C07319=1203.614,129.321,-51.756,-178.380,5.980,148.587
C07320=1203.610,129.570,-51.775,-178.377,5.982,148.587
C07321=1203.605,129.819,-51.796,-178.374,5.982,148.586
C07322=1203.600,130.069,-51.815,-178.372,5.984,148.586
C07323=1203.596,130.318,-51.836,-178.370,5.985,148.585
C07324=1203.591,130.567,-51.855,-178.366,5.986,148.585
C07325=1203.586,130.816,-51.875,-178.364,5.988,148.584
C07326=1203.581,131.065,-51.896,-178.361,5.989,148.584
C07327=1203.576,131.315,-51.916,-178.358,5.991,148.583
C07328=1203.572,131.563,-51.936,-178.356,5.992,148.583
C07329=1203.567,131.813,-51.956,-178.353,5.993,148.582
C07330=1203.563,132.062,-51.976,-178.351,5.994,148.582
C07331=1203.558,132.311,-51.997,-178.348,5.996,148.581
C07332=1203.552,132.560,-52.017,-178.346,5.996,148.581
C07333=1203.548,132.828,-52.039,-178.343,5.998,148.580
C07334=1203.542,133.098,-52.061,-178.340,5.999,148.580
C07335=1203.538,133.366,-52.082,-178.337,6.001,148.579
C07336=1203.532,133.635,-52.104,-178.334,6.003,148.579
C07337=1203.528,133.884,-52.124,-178.332,6.004,148.578
C07338=1203.523,134.133,-52.144,-178.329,6.005,148.578
C07339=1203.519,134.382,-52.164,-178.327,6.006,148.577
C07340=1203.513,134.631,-52.185,-178.324,6.008,148.577
C07341=1203.508,134.880,-52.205,-178.321,6.008,148.576
C07342=1203.504,135.129,-52.225,-178.319,6.010,148.576
C07343=1203.499,135.378,-52.245,-178.316,6.012,148.576
C07344=1203.494,135.628,-52.266,-178.313,6.013,148.575
C07345=1203.489,135.877,-52.286,-178.311,6.014,148.575
C07346=1203.485,136.126,-52.306,-178.309,6.015,148.574
C07347=1203.480,136.375,-52.327,-178.305,6.017,148.574
C07348=1203.475,136.624,-52.348,-178.303,6.018,148.573
C07349=1203.471,136.873,-52.368,-178.301,6.019,148.573
C07350=1203.466,137.123,-52.388,-178.297,6.021,148.572
C07351=1203.461,137.372,-52.409,-178.295,6.022,148.572
C07352=1203.456,137.621,-52.429,-178.293,6.024,148.571
C07353=1203.452,137.870,-52.450,-178.290,6.024,148.571
C07354=1203.447,138.119,-52.470,-178.287,6.026,148.570
C07355=1203.442,138.367,-52.490,-178.285,6.028,148.570
C07356=1203.437,138.616,-52.511,-178.282,6.028,148.569
C07357=1203.432,138.866,-52.531,-178.279,6.030,148.569
C07358=1203.427,139.115,-52.551,-178.277,6.031,148.569
C07359=1203.423,139.364,-52.572,-178.274,6.033,148.568
C07360=1203.418,139.613,-52.593,-178.271,6.034,148.568
C07361=1203.413,139.862,-52.613,-178.269,6.035,148.567
C07362=1203.408,140.112,-52.634,-178.266,6.037,148.567
C07363=1203.404,140.361,-52.655,-178.264,6.038,148.566
C07364=1203.399,140.610,-52.675,-178.261,6.040,148.566
C07365=1203.394,140.859,-52.696,-178.258,6.041,148.565
C07366=1203.390,141.108,-52.716,-178.256,6.042,148.565
C07367=1203.385,141.357,-52.737,-178.253,6.044,148.564
C07368=1203.381,141.607,-52.758,-178.251,6.046,148.564
C07369=1203.376,141.856,-52.778,-178.248,6.046,148.563
C07370=1203.371,142.105,-52.799,-178.245,6.048,148.563
C07371=1203.367,142.354,-52.820,-178.243,6.049,148.563
C07372=1203.362,142.603,-52.841,-178.240,6.050,148.562
C07373=1203.357,142.852,-52.861,-178.237,6.052,148.562
C07374=1203.352,143.101,-52.882,-178.235,6.053,148.561
C07375=1203.347,143.350,-52.902,-178.232,6.054,148.561
C07376=1203.342,143.599,-52.923,-178.229,6.056,148.560
C07377=1203.338,143.848,-52.944,-178.227,6.057,148.560
C07378=1203.333,144.098,-52.965,-178.225,6.059,148.559
C07379=1203.328,144.347,-52.985,-178.222,6.060,148.559
C07380=1203.323,144.595,-53.007,-178.219,6.061,148.558
C07381=1203.319,144.844,-53.027,-178.217,6.063,148.558
C07382=1203.314,145.093,-53.048,-178.214,6.064,148.557
C07383=1203.309,145.342,-53.068,-178.211,6.066,148.557
C07384=1203.305,145.592,-53.090,-178.209,6.067,148.557
C07385=1203.300,145.841,-53.110,-178.207,6.068,148.556
C07386=1203.295,146.091,-53.131,-178.204,6.070,148.556
C07387=1203.291,146.339,-53.152,-178.201,6.072,148.555
C07388=1203.286,146.588,-53.173,-178.199,6.073,148.555
C07389=1203.281,146.837,-53.193,-178.196,6.074,148.554
C07390=1203.276,147.086,-53.214,-178.193,6.076,148.554
C07391=1203.271,147.335,-53.236,-178.191,6.077,148.553
C07392=1203.268,147.585,-53.257,-178.188,6.079,148.553
C07393=1203.262,147.834,-53.278,-178.185,6.079,148.552
C07394=1203.258,148.083,-53.298,-178.183,6.081,148.552
C07395=1203.253,148.332,-53.320,-178.180,6.083,148.552
C07396=1203.248,148.581,-53.341,-178.178,6.084,148.551
C07397=1203.243,148.830,-53.361,-178.175,6.085,148.551
C07398=1203.238,149.079,-53.382,-178.172,6.087,148.550
C07399=1203.234,149.328,-53.404,-178.170,6.088,148.550
C07400=1203.230,149.577,-53.425,-178.167,6.090,148.550
C07401=1203.224,149.827,-53.446,-178.164,6.091,148.549
C07402=1203.219,150.075,-53.467,-178.162,6.092,148.549
C07403=1203.215,150.324,-53.488,-178.159,6.094,148.548
C07404=1203.210,150.573,-53.509,-178.157,6.096,148.548
C07405=1203.206,150.823,-53.531,-178.154,6.097,148.547
C07406=1203.201,151.072,-53.551,-178.151,6.098,148.547
C07407=1203.196,151.320,-53.573,-178.149,6.100,148.546
C07408=1203.191,151.570,-53.594,-178.146,6.102,148.546
C07409=1203.187,151.819,-53.614,-178.144,6.102,148.545
C07410=1203.182,152.068,-53.636,-178.141,6.104,148.545
C07411=1203.177,152.317,-53.657,-178.138,6.106,148.545
C07412=1203.172,152.566,-53.679,-178.136,6.107,148.544
C07413=1203.168,152.815,-53.699,-178.133,6.108,148.544
C07414=1203.163,153.063,-53.721,-178.130,6.110,148.543
C07415=1203.159,153.313,-53.742,-178.128,6.111,148.543
C07416=1203.154,153.562,-53.764,-178.125,6.113,148.543
C07417=1203.149,153.811,-53.784,-178.122,6.114,148.542
C07418=1203.144,154.060,-53.805,-178.120,6.115,148.542
C07419=1203.140,154.310,-53.827,-178.118,6.117,148.541
C07420=1203.135,154.558,-53.849,-178.115,6.119,148.541
C07421=1203.130,154.807,-53.869,-178.112,6.120,148.540
C07422=1203.126,155.056,-53.891,-178.110,6.121,148.540
C07423=1203.121,155.306,-53.912,-178.107,6.123,148.539
C07424=1203.116,155.554,-53.934,-178.104,6.125,148.539
C07425=1203.111,155.804,-53.955,-178.102,6.126,148.539
C07426=1203.107,156.053,-53.977,-178.099,6.127,148.538
C07427=1203.102,156.302,-53.997,-178.096,6.129,148.538
C07428=1203.097,156.551,-54.019,-178.094,6.131,148.537
C07429=1203.093,156.799,-54.041,-178.092,6.132,148.537
C07430=1203.088,157.049,-54.062,-178.089,6.134,148.537
C07431=1203.083,157.298,-54.084,-178.086,6.135,148.536
C07432=1203.078,157.546,-54.105,-178.084,6.136,148.536
C07433=1203.074,157.796,-54.127,-178.081,6.138,148.535
C07434=1203.070,158.045,-54.148,-178.078,6.140,148.535
C07435=1203.065,158.293,-54.170,-178.075,6.141,148.534
C07436=1203.060,158.543,-54.191,-178.073,6.142,148.534
C07437=1203.055,158.812,-54.215,-178.070,6.144,148.533
C07438=1203.050,159.080,-54.237,-178.068,6.146,148.533
C07439=1203.044,159.350,-54.261,-178.064,6.147,148.533
C07440=1203.040,159.618,-54.284,-178.062,6.149,148.532
C07441=1203.035,159.868,-54.305,-178.059,6.151,148.532
C07442=1203.030,160.117,-54.327,-178.056,6.152,148.531
C07443=1203.025,160.365,-54.349,-178.054,6.153,148.531
C07444=1203.021,160.615,-54.371,-178.051,6.155,148.530
C07445=1203.016,160.864,-54.392,-178.049,6.157,148.530
C07446=1203.012,161.113,-54.414,-178.046,6.158,148.530
C07447=1203.007,161.362,-54.436,-178.043,6.159,148.529
C07448=1203.002,161.611,-54.457,-178.041,6.161,148.529
C07449=1202.998,161.860,-54.479,-178.038,6.163,148.528
C07450=1202.992,162.109,-54.500,-178.035,6.164,148.528
C07451=1202.988,162.359,-54.522,-178.033,6.165,148.528
C07452=1202.983,162.607,-54.544,-178.030,6.167,148.527
C07453=1202.978,162.856,-54.566,-178.027,6.169,148.527
C07454=1202.974,163.105,-54.588,-178.025,6.170,148.526
C07455=1202.969,163.354,-54.609,-178.023,6.171,148.526
C07456=1202.965,163.603,-54.631,-178.020,6.173,148.525
C07457=1202.960,163.852,-54.653,-178.017,6.175,148.525
C07458=1202.955,164.100,-54.675,-178.015,6.177,148.525
C07459=1202.951,164.350,-54.696,-178.012,6.177,148.524
C07460=1202.946,164.599,-54.718,-178.009,6.179,148.524
C07461=1202.942,164.848,-54.740,-178.007,6.181,148.523
C07462=1202.936,165.097,-54.762,-178.004,6.183,148.523
C07463=1202.932,165.347,-54.784,-178.002,6.184,148.523
C07464=1202.927,165.595,-54.806,-177.999,6.186,148.522
C07465=1202.923,165.845,-54.828,-177.996,6.187,148.522
C07466=1202.918,166.093,-54.850,-177.993,6.189,148.521
C07467=1202.913,166.342,-54.871,-177.991,6.191,148.521
C07468=1202.909,166.591,-54.893,-177.989,6.192,148.521
C07469=1202.904,166.840,-54.915,-177.986,6.193,148.520
C07470=1202.899,167.089,-54.937,-177.983,6.195,148.520
C07471=1202.894,167.338,-54.959,-177.981,6.197,148.519
C07472=1202.890,167.587,-54.982,-177.978,6.198,148.519
C07473=1202.885,167.836,-55.004,-177.975,6.199,148.518
C07474=1202.881,168.085,-55.026,-177.973,6.201,148.518
C07475=1202.876,168.334,-55.048,-177.970,6.203,148.518
C07476=1202.872,168.583,-55.070,-177.967,6.205,148.517
C07477=1202.866,168.832,-55.092,-177.965,6.206,148.517
C07478=1202.862,169.081,-55.114,-177.963,6.208,148.517
C07479=1202.857,169.330,-55.136,-177.959,6.209,148.516
C07480=1202.853,169.579,-55.158,-177.957,6.211,148.516
C07481=1202.848,169.827,-55.180,-177.954,6.213,148.515
C07482=1202.843,170.077,-55.203,-177.952,6.214,148.515
C07483=1202.838,170.326,-55.224,-177.949,6.215,148.515
C07484=1202.834,170.575,-55.246,-177.947,6.217,148.514
C07485=1202.830,170.824,-55.268,-177.944,6.219,148.514
C07486=1202.824,171.073,-55.291,-177.941,6.221,148.513
C07487=1202.820,171.322,-55.314,-177.939,6.222,148.513
C07488=1202.815,171.571,-55.335,-177.936,6.223,148.513
C07489=1202.810,171.820,-55.358,-177.933,6.225,148.512
C07490=1202.806,172.068,-55.380,-177.931,6.227,148.512
C07491=1202.801,172.318,-55.402,-177.928,6.229,148.511
C07492=1202.796,172.566,-55.424,-177.925,6.231,148.511
C07493=1202.791,172.816,-55.447,-177.923,6.232,148.511
C07494=1202.787,173.065,-55.469,-177.921,6.233,148.510
C07495=1202.783,173.313,-55.491,-177.918,6.235,148.510
C07496=1202.778,173.563,-55.514,-177.915,6.237,148.509
C07497=1202.773,173.811,-55.536,-177.912,6.238,148.509
C07498=1202.769,174.060,-55.558,-177.909,6.240,148.509
C07499=1202.764,174.310,-55.581,-177.907,6.241,148.508
C07500=1202.759,174.558,-55.603,-177.905,6.243,148.508
C07501=1202.755,174.807,-55.625,-177.902,6.245,148.508
C07502=1202.749,175.056,-55.648,-177.899,6.247,148.507
C07503=1202.745,175.305,-55.670,-177.897,6.248,148.507
C07504=1202.740,175.555,-55.693,-177.894,6.250,148.506
C07505=1202.736,175.803,-55.715,-177.892,6.251,148.506
C07506=1202.732,176.052,-55.737,-177.889,6.253,148.506
C07507=1202.727,176.301,-55.761,-177.886,6.254,148.505
C07508=1202.722,176.550,-55.782,-177.883,6.256,148.505
C07509=1202.717,176.799,-55.805,-177.881,6.258,148.504
C07510=1202.713,177.048,-55.828,-177.878,6.260,148.504
C07511=1202.708,177.297,-55.850,-177.876,6.261,148.504
C07512=1202.703,177.546,-55.873,-177.873,6.263,148.503
C07513=1202.699,177.795,-55.895,-177.871,6.264,148.503
C07514=1202.694,178.043,-55.918,-177.868,6.266,148.503
C07515=1202.690,178.293,-55.940,-177.865,6.268,148.502
C07516=1202.685,178.542,-55.963,-177.863,6.270,148.502
C07517=1202.680,178.790,-55.986,-177.860,6.272,148.502
C07518=1202.675,179.039,-56.008,-177.858,6.273,148.501
C07519=1202.671,179.288,-56.031,-177.855,6.274,148.501
C07520=1202.666,179.537,-56.053,-177.852,6.276,148.500
C07521=1202.662,179.786,-56.076,-177.849,6.278,148.500
C07522=1202.657,180.035,-56.099,-177.847,6.280,148.499
C07523=1202.653,180.284,-56.122,-177.844,6.281,148.499
C07524=1202.647,180.532,-56.145,-177.841,6.283,148.499
C07525=1202.643,180.782,-56.167,-177.839,6.285,148.498
C07526=1202.639,181.031,-56.190,-177.837,6.286,148.498
C07527=1202.635,181.280,-56.213,-177.834,6.288,148.498
C07528=1202.629,181.528,-56.235,-177.831,6.290,148.497
C07529=1202.625,181.777,-56.258,-177.829,6.291,148.497
C07530=1202.620,182.026,-56.281,-177.826,6.293,148.497
C07531=1202.615,182.276,-56.304,-177.823,6.295,148.496
C07532=1202.611,182.524,-56.326,-177.821,6.297,148.496
C07533=1202.606,182.773,-56.350,-177.818,6.299,148.496
C07534=1202.602,183.022,-56.372,-177.815,6.300,148.495
C07535=1202.597,183.271,-56.395,-177.813,6.301,148.495
C07536=1202.592,183.519,-56.417,-177.811,6.303,148.494
C07537=1202.588,183.768,-56.441,-177.808,6.305,148.494
C07538=1202.583,184.017,-56.464,-177.805,6.307,148.494
C07539=1202.579,184.267,-56.486,-177.803,6.309,148.493
C07540=1202.574,184.516,-56.509,-177.800,6.310,148.493
C07541=1202.569,184.786,-56.535,-177.797,6.312,148.492
C07542=1202.564,185.055,-56.559,-177.794,6.314,148.492
C07543=1202.559,185.325,-56.584,-177.792,6.316,148.492
C07544=1202.554,185.594,-56.608,-177.789,6.317,148.491
C07545=1202.549,185.843,-56.631,-177.786,6.319,148.491
C07546=1202.544,186.092,-56.655,-177.784,6.321,148.491
C07547=1202.540,186.341,-56.678,-177.781,6.323,148.490
C07548=1202.536,186.589,-56.701,-177.778,6.325,148.490
C07549=1202.531,186.838,-56.724,-177.776,6.326,148.490
C07550=1202.526,187.087,-56.748,-177.773,6.328,148.489
C07551=1202.522,187.335,-56.770,-177.770,6.330,148.489
C07552=1202.517,187.584,-56.793,-177.768,6.332,148.489
C07553=1202.512,187.834,-56.816,-177.765,6.334,148.488
C07554=1202.507,188.083,-56.839,-177.762,6.335,148.488
C07555=1202.503,188.332,-56.862,-177.760,6.337,148.488
C07556=1202.499,188.581,-56.886,-177.758,6.338,148.487
C07557=1202.494,188.830,-56.909,-177.755,6.340,148.487
C07558=1202.489,189.078,-56.932,-177.752,6.342,148.486
C07559=1202.485,189.327,-56.955,-177.750,6.344,148.486
C07560=1202.480,189.576,-56.978,-177.747,6.346,148.486
C07561=1202.475,189.825,-57.001,-177.744,6.347,148.485
C07562=1202.471,190.074,-57.025,-177.742,6.349,148.485
C07563=1202.466,190.323,-57.048,-177.739,6.351,148.485
C07564=1202.461,190.572,-57.071,-177.736,6.353,148.484
C07565=1202.458,190.820,-57.095,-177.734,6.355,148.484
C07566=1202.453,191.069,-57.118,-177.731,6.356,148.484
C07567=1202.448,191.318,-57.141,-177.728,6.358,148.483
C07568=1202.443,191.567,-57.165,-177.726,6.360,148.483
C07569=1202.438,191.816,-57.188,-177.723,6.362,148.483
C07570=1202.433,192.065,-57.211,-177.720,6.364,148.482
C07571=1202.429,192.313,-57.234,-177.718,6.365,148.482
C07572=1202.425,192.562,-57.257,-177.715,6.367,148.482
C07573=1202.420,192.811,-57.281,-177.712,6.369,148.481
C07574=1202.416,193.060,-57.305,-177.710,6.370,148.481
C07575=1202.411,193.309,-57.328,-177.708,6.372,148.480
C07576=1202.406,193.558,-57.352,-177.705,6.374,148.480
C07577=1202.402,193.807,-57.375,-177.702,6.376,148.480
C07578=1202.397,194.056,-57.398,-177.700,6.377,148.479
C07579=1202.392,194.304,-57.422,-177.697,6.379,148.479
C07580=1202.388,194.553,-57.446,-177.694,6.381,148.479
C07581=1202.383,194.802,-57.469,-177.692,6.383,148.478
C07582=1202.378,195.052,-57.492,-177.689,6.385,148.478
C07583=1202.374,195.300,-57.517,-177.686,6.386,148.478
C07584=1202.369,195.549,-57.540,-177.684,6.388,148.477
C07585=1202.365,195.798,-57.563,-177.681,6.390,148.477
C07586=1202.361,196.047,-57.586,-177.678,6.392,148.477
C07587=1202.356,196.295,-57.610,-177.676,6.394,148.476
C07588=1202.352,196.544,-57.633,-177.673,6.396,148.476
C07589=1202.347,196.793,-57.657,-177.671,6.397,148.476
C07590=1202.342,197.042,-57.681,-177.668,6.399,148.475
C07591=1202.338,197.291,-57.704,-177.665,6.401,148.475
C07592=1202.332,197.540,-57.728,-177.663,6.403,148.475
C07593=1202.328,197.788,-57.752,-177.660,6.405,148.474
C07594=1202.323,198.037,-57.776,-177.658,6.407,148.474
C07595=1202.319,198.286,-57.800,-177.655,6.409,148.474
C07596=1202.314,198.535,-57.823,-177.652,6.410,148.473
C07597=1202.309,198.784,-57.846,-177.650,6.412,148.473
C07598=1202.305,199.032,-57.870,-177.647,6.414,148.473
C07599=1202.300,199.281,-57.894,-177.644,6.416,148.472
C07600=1202.296,199.530,-57.918,-177.642,6.418,148.472
C07601=1202.291,199.779,-57.941,-177.639,6.420,148.472
C07602=1202.287,200.027,-57.965,-177.637,6.421,148.471
C07603=1202.283,200.277,-57.989,-177.634,6.423,148.471
C07604=1202.278,200.525,-58.013,-177.631,6.425,148.471
C07605=1202.273,200.775,-58.037,-177.629,6.427,148.470
C07606=1202.268,201.023,-58.061,-177.626,6.429,148.470
C07607=1202.264,201.272,-58.085,-177.624,6.431,148.470
C07608=1202.259,201.521,-58.109,-177.621,6.433,148.469
C07609=1202.255,201.770,-58.132,-177.618,6.434,148.469
C07610=1202.250,202.018,-58.156,-177.616,6.436,148.469
C07611=1202.246,202.267,-58.179,-177.613,6.438,148.468
C07612=1202.240,202.516,-58.204,-177.610,6.440,148.468
C07613=1202.237,202.765,-58.229,-177.608,6.442,148.468
C07614=1202.232,203.014,-58.252,-177.605,6.444,148.467
C07615=1202.228,203.262,-58.276,-177.603,6.445,148.467
C07616=1202.223,203.511,-58.300,-177.600,6.447,148.467
C07617=1202.218,203.760,-58.324,-177.597,6.449,148.466
C07618=1202.213,204.008,-58.348,-177.595,6.451,148.466
C07619=1202.209,204.258,-58.372,-177.592,6.453,148.466
C07620=1202.205,204.507,-58.396,-177.590,6.455,148.466
C07621=1202.200,204.755,-58.420,-177.587,6.457,148.465
C07622=1202.195,205.004,-58.445,-177.584,6.458,148.465
C07623=1202.191,205.253,-58.468,-177.582,6.460,148.465
C07624=1202.186,205.501,-58.492,-177.579,6.462,148.464
C07625=1202.182,205.750,-58.516,-177.576,6.465,148.464
C07626=1202.177,206.000,-58.540,-177.573,6.467,148.464
C07627=1202.173,206.248,-58.565,-177.571,6.469,148.463
C07628=1202.168,206.496,-58.589,-177.568,6.471,148.463
C07629=1202.163,206.745,-58.613,-177.566,6.472,148.463
C07630=1202.159,206.995,-58.637,-177.563,6.474,148.462
C07631=1202.155,207.243,-58.661,-177.561,6.476,148.462
C07632=1202.149,207.492,-58.686,-177.558,6.478,148.462
C07633=1202.145,207.741,-58.710,-177.555,6.480,148.461
C07634=1202.141,207.989,-58.734,-177.553,6.481,148.461
C07635=1202.136,208.238,-58.759,-177.550,6.484,148.461
C07636=1202.131,208.487,-58.782,-177.548,6.485,148.461
C07637=1202.127,208.736,-58.806,-177.545,6.487,148.460
C07638=1202.122,208.985,-58.831,-177.542,6.489,148.460
C07639=1202.118,209.234,-58.855,-177.540,6.491,148.460
C07640=1202.114,209.482,-58.880,-177.537,6.493,148.459
C07641=1202.109,209.731,-58.904,-177.535,6.495,148.459
C07642=1202.104,209.979,-58.928,-177.532,6.498,148.459
C07643=1202.100,210.229,-58.953,-177.529,6.499,148.459
C07644=1202.095,210.477,-58.977,-177.527,6.501,148.458
C07645=1202.090,210.748,-59.003,-177.524,6.503,148.458
C07646=1202.085,211.018,-59.030,-177.521,6.505,148.458
C07647=1202.080,211.289,-59.057,-177.518,6.508,148.457
C07648=1202.076,211.559,-59.083,-177.515,6.509,148.457
C07649=1202.071,211.807,-59.108,-177.513,6.511,148.457
C07650=1202.066,212.056,-59.132,-177.510,6.513,148.456
C07651=1202.062,212.305,-59.157,-177.507,6.515,148.456
C07652=1202.057,212.554,-59.181,-177.505,6.517,148.456
C07653=1202.052,212.802,-59.206,-177.502,6.520,148.455
C07654=1202.048,213.052,-59.230,-177.499,6.521,148.455
C07655=1202.043,213.300,-59.255,-177.497,6.523,148.455
C07656=1202.039,213.549,-59.279,-177.494,6.525,148.454
C07657=1202.034,213.798,-59.304,-177.491,6.527,148.454
C07658=1202.030,214.046,-59.328,-177.489,6.529,148.454
C07659=1202.025,214.295,-59.353,-177.487,6.531,148.454
C07660=1202.021,214.544,-59.378,-177.484,6.533,148.453
C07661=1202.016,214.792,-59.403,-177.481,6.535,148.453
C07662=1202.012,215.041,-59.427,-177.479,6.536,148.453
C07663=1202.007,215.290,-59.452,-177.476,6.539,148.452
C07664=1202.002,215.539,-59.476,-177.473,6.541,148.452
C07665=1201.998,215.788,-59.501,-177.471,6.543,148.452
C07666=1201.993,216.036,-59.526,-177.468,6.545,148.452
C07667=1201.989,216.285,-59.550,-177.465,6.547,148.451
C07668=1201.985,216.534,-59.575,-177.463,6.549,148.451
C07669=1201.980,216.782,-59.599,-177.460,6.550,148.451
C07670=1201.975,217.031,-59.624,-177.458,6.553,148.450
C07671=1201.971,217.280,-59.650,-177.455,6.554,148.450
C07672=1201.966,217.528,-59.674,-177.452,6.557,148.450
C07673=1201.962,217.778,-59.699,-177.449,6.559,148.449
C07674=1201.957,218.026,-59.724,-177.447,6.561,148.449
C07675=1201.953,218.274,-59.748,-177.445,6.563,148.449
C07676=1201.948,218.524,-59.773,-177.442,6.565,148.449
C07677=1201.943,218.772,-59.798,-177.439,6.567,148.448
C07678=1201.939,219.021,-59.823,-177.437,6.568,148.448
C07679=1201.934,219.270,-59.848,-177.434,6.570,148.448
C07680=1201.930,219.519,-59.873,-177.431,6.573,148.448
C07681=1201.926,219.767,-59.898,-177.429,6.575,148.447
C07682=1201.921,220.016,-59.923,-177.426,6.577,148.447
C07683=1201.916,220.264,-59.948,-177.423,6.579,148.447
C07684=1201.913,220.514,-59.973,-177.421,6.581,148.446
C07685=1201.907,220.762,-59.997,-177.419,6.583,148.446
C07686=1201.903,221.010,-60.023,-177.416,6.584,148.446
C07687=1201.898,221.260,-60.048,-177.413,6.586,148.446
C07688=1201.894,221.508,-60.072,-177.410,6.589,148.445
C07689=1201.889,221.757,-60.097,-177.408,6.591,148.445
C07690=1201.885,222.005,-60.123,-177.405,6.593,148.445
C07691=1201.880,222.255,-60.148,-177.403,6.595,148.444
C07692=1201.876,222.502,-60.173,-177.400,6.597,148.444
C07693=1201.872,222.752,-60.198,-177.398,6.599,148.444
C07694=1201.867,223.000,-60.223,-177.395,6.601,148.444
C07695=1201.862,223.249,-60.248,-177.392,6.603,148.443
C07696=1201.857,223.497,-60.274,-177.389,6.605,148.443
C07697=1201.854,223.747,-60.298,-177.387,6.607,148.443
C07698=1201.849,223.995,-60.323,-177.385,6.609,148.443
C07699=1201.844,224.244,-60.348,-177.382,6.611,148.442
C07700=1201.840,224.493,-60.374,-177.379,6.613,148.442
C07701=1201.835,224.741,-60.400,-177.377,6.616,148.442
C07702=1201.831,224.990,-60.425,-177.374,6.618,148.442
C07703=1201.827,225.238,-60.449,-177.371,6.619,148.441
C07704=1201.822,225.488,-60.474,-177.369,6.621,148.441
C07705=1201.817,225.736,-60.500,-177.367,6.623,148.441
C07706=1201.813,225.984,-60.526,-177.364,6.625,148.441
C07707=1201.808,226.233,-60.550,-177.361,6.627,148.440
C07708=1201.804,226.482,-60.576,-177.358,6.630,148.440
C07709=1201.799,226.731,-60.602,-177.356,6.632,148.440
C07710=1201.794,226.980,-60.626,-177.353,6.634,148.439
C07711=1201.790,227.228,-60.652,-177.351,6.636,148.439
C07712=1201.786,227.476,-60.677,-177.348,6.638,148.439
C07713=1201.782,227.725,-60.703,-177.346,6.640,148.439
C07714=1201.777,227.974,-60.728,-177.343,6.642,148.438
C07715=1201.772,228.222,-60.753,-177.340,6.644,148.438
C07716=1201.768,228.471,-60.779,-177.338,6.646,148.438
C07717=1201.763,228.719,-60.804,-177.335,6.648,148.438
C07718=1201.759,228.969,-60.829,-177.333,6.650,148.437
C07719=1201.755,229.218,-60.855,-177.330,6.653,148.437
C07720=1201.750,229.466,-60.880,-177.327,6.655,148.437
C07721=1201.745,229.715,-60.906,-177.325,6.657,148.437
C07722=1201.741,229.963,-60.932,-177.322,6.659,148.437
C07723=1201.736,230.212,-60.957,-177.320,6.661,148.436
C07724=1201.732,230.461,-60.982,-177.317,6.662,148.436
C07725=1201.727,230.709,-61.008,-177.314,6.665,148.436
C07726=1201.723,230.958,-61.033,-177.312,6.667,148.435
C07727=1201.719,231.207,-61.059,-177.309,6.669,148.435
C07728=1201.714,231.455,-61.085,-177.307,6.671,148.435
C07729=1201.710,231.703,-61.110,-177.304,6.673,148.435
C07730=1201.705,231.952,-61.136,-177.301,6.676,148.434
C07731=1201.700,232.201,-61.162,-177.299,6.678,148.434
C07732=1201.696,232.450,-61.188,-177.296,6.680,148.434
C07733=1201.691,232.699,-61.213,-177.294,6.682,148.434
C07734=1201.687,232.948,-61.239,-177.291,6.683,148.433
C07735=1201.682,233.196,-61.264,-177.288,6.686,148.433
C07736=1201.678,233.445,-61.290,-177.286,6.688,148.433
C07737=1201.674,233.693,-61.316,-177.283,6.690,148.433
C07738=1201.669,233.942,-61.341,-177.281,6.692,148.433
C07739=1201.664,234.190,-61.367,-177.278,6.694,148.432
C07740=1201.660,234.439,-61.394,-177.275,6.697,148.432
C07741=1201.655,234.687,-61.419,-177.273,6.699,148.432
C07742=1201.651,234.936,-61.445,-177.270,6.701,148.432
C07743=1201.647,235.185,-61.471,-177.268,6.703,148.431
C07744=1201.642,235.433,-61.496,-177.266,6.705,148.431
C07745=1201.637,235.681,-61.522,-177.262,6.708,148.431
C07746=1201.633,235.931,-61.548,-177.260,6.710,148.431
C07747=1201.628,236.179,-61.574,-177.258,6.712,148.430
C07748=1201.624,236.428,-61.600,-177.255,6.713,148.430
C07749=1201.619,236.699,-61.628,-177.252,6.716,148.430
C07750=1201.614,236.971,-61.656,-177.250,6.718,148.430
C07751=1201.610,237.243,-61.684,-177.246,6.721,148.429
C07752=1201.604,237.513,-61.713,-177.244,6.723,148.429
C07753=1201.600,237.762,-61.739,-177.241,6.726,148.429
C07754=1201.596,238.011,-61.765,-177.238,6.728,148.429
C07755=1201.591,238.260,-61.790,-177.236,6.729,148.428
C07756=1201.587,238.508,-61.817,-177.234,6.732,148.428
C07757=1201.582,238.756,-61.843,-177.230,6.734,148.428
C07758=1201.578,239.005,-61.868,-177.228,6.736,148.428
C07759=1201.573,239.254,-61.894,-177.226,6.738,148.428
C07760=1201.569,239.503,-61.921,-177.223,6.740,148.427
C07761=1201.564,239.751,-61.947,-177.221,6.742,148.427
C07762=1201.560,239.999,-61.972,-177.218,6.745,148.427
C07763=1201.555,240.248,-61.999,-177.215,6.747,148.427
C07764=1201.551,240.497,-62.025,-177.213,6.749,148.426
C07765=1201.547,240.746,-62.051,-177.210,6.751,148.426
C07766=1201.542,240.994,-62.078,-177.207,6.754,148.426
C07767=1201.538,241.243,-62.104,-177.205,6.756,148.426
C07768=1201.533,241.491,-62.129,-177.203,6.758,148.426
C07769=1201.528,241.739,-62.156,-177.200,6.760,148.425
C07770=1201.524,241.988,-62.182,-177.197,6.762,148.425
C07771=1201.519,242.237,-62.208,-177.195,6.764,148.425
C07772=1201.515,242.486,-62.235,-177.192,6.766,148.425
C07773=1201.511,242.734,-62.261,-177.189,6.769,148.425
C07774=1201.506,242.983,-62.288,-177.187,6.771,148.424
C07775=1201.502,243.232,-62.313,-177.184,6.773,148.424
C07776=1201.497,243.480,-62.340,-177.182,6.775,148.424
C07777=1201.492,243.728,-62.366,-177.179,6.778,148.424
C07778=1201.489,243.976,-62.392,-177.177,6.780,148.423
C07779=1201.484,244.226,-62.419,-177.174,6.782,148.423
C07780=1201.480,244.474,-62.445,-177.172,6.784,148.423
C07781=1201.475,244.723,-62.471,-177.169,6.787,148.423
C07782=1201.471,244.971,-62.498,-177.166,6.789,148.422
C07783=1201.466,245.220,-62.524,-177.164,6.791,148.422
C07784=1201.462,245.468,-62.551,-177.161,6.793,148.422
C07785=1201.457,245.718,-62.577,-177.159,6.796,148.422
C07786=1201.453,245.966,-62.604,-177.156,6.797,148.422
C07787=1201.448,246.214,-62.631,-177.154,6.800,148.422
C07788=1201.444,246.463,-62.656,-177.151,6.802,148.421
C07789=1201.440,246.711,-62.683,-177.148,6.804,148.421
C07790=1201.435,246.960,-62.709,-177.146,6.806,148.421
C07791=1201.430,247.208,-62.736,-177.143,6.809,148.421
C07792=1201.426,247.456,-62.762,-177.140,6.811,148.421
C07793=1201.421,247.705,-62.789,-177.138,6.813,148.420
C07794=1201.417,247.954,-62.815,-177.136,6.815,148.420
C07795=1201.413,248.202,-62.842,-177.132,6.818,148.420
C07796=1201.408,248.451,-62.869,-177.130,6.820,148.420
C07797=1201.404,248.699,-62.895,-177.128,6.822,148.419
C07798=1201.399,248.948,-62.922,-177.125,6.825,148.419
C07799=1201.395,249.197,-62.948,-177.122,6.827,148.419
C07800=1201.390,249.445,-62.975,-177.120,6.829,148.419
C07801=1201.385,249.694,-63.002,-177.117,6.832,148.419
C07802=1201.382,249.942,-63.028,-177.115,6.834,148.419
C07803=1201.377,250.190,-63.055,-177.112,6.836,148.418
C07804=1201.373,250.439,-63.081,-177.110,6.838,148.418
C07805=1201.368,250.688,-63.108,-177.107,6.840,148.418
C07806=1201.363,250.936,-63.135,-177.105,6.843,148.418
C07807=1201.360,251.185,-63.162,-177.102,6.844,148.418
C07808=1201.355,251.434,-63.189,-177.099,6.847,148.418
C07809=1201.350,251.683,-63.216,-177.097,6.849,148.417
C07810=1201.347,251.931,-63.242,-177.095,6.851,148.417
C07811=1201.342,252.179,-63.269,-177.091,6.854,148.417
C07812=1201.337,252.428,-63.296,-177.089,6.856,148.417
C07813=1201.333,252.676,-63.323,-177.087,6.858,148.416
C07814=1201.329,252.924,-63.350,-177.084,6.861,148.416
C07815=1201.324,253.173,-63.377,-177.081,6.863,148.416
C07816=1201.319,253.421,-63.404,-177.079,6.865,148.416
C07817=1201.315,253.670,-63.430,-177.076,6.868,148.416
C07818=1201.311,253.918,-63.457,-177.074,6.870,148.416
C07819=1201.306,254.167,-63.484,-177.071,6.872,148.415
C07820=1201.301,254.415,-63.511,-177.068,6.875,148.415
C07821=1201.298,254.664,-63.538,-177.066,6.877,148.415
C07822=1201.293,254.913,-63.565,-177.064,6.879,148.415
C07823=1201.289,255.161,-63.592,-177.061,6.882,148.415
C07824=1201.284,255.410,-63.619,-177.058,6.884,148.415
C07825=1201.279,255.658,-63.647,-177.056,6.886,148.414
C07826=1201.276,255.906,-63.673,-177.053,6.889,148.414
C07827=1201.271,256.155,-63.700,-177.051,6.891,148.414
C07828=1201.266,256.403,-63.727,-177.048,6.894,148.414
C07829=1201.262,256.652,-63.755,-177.046,6.896,148.414
C07830=1201.258,256.901,-63.782,-177.043,6.898,148.413
C07831=1201.253,257.149,-63.809,-177.040,6.901,148.413
C07832=1201.249,257.398,-63.835,-177.038,6.902,148.413
C07833=1201.244,257.646,-63.862,-177.035,6.905,148.413
C07834=1201.240,257.895,-63.889,-177.032,6.907,148.413
C07835=1201.236,258.143,-63.917,-177.030,6.909,148.413
C07836=1201.231,258.392,-63.944,-177.028,6.912,148.413
C07837=1201.227,258.640,-63.972,-177.025,6.914,148.412
C07838=1201.222,258.889,-63.999,-177.023,6.916,148.412
C07839=1201.217,259.137,-64.026,-177.019,6.919,148.412
C07840=1201.214,259.385,-64.053,-177.017,6.921,148.412
C07841=1201.210,259.634,-64.080,-177.015,6.923,148.412
C07842=1201.205,259.882,-64.107,-177.012,6.926,148.411
C07843=1201.200,260.131,-64.134,-177.010,6.928,148.411
C07844=1201.196,260.379,-64.162,-177.007,6.930,148.411
C07845=1201.192,260.628,-64.190,-177.004,6.933,148.411
C07846=1201.187,260.876,-64.217,-177.002,6.935,148.411
C07847=1201.183,261.125,-64.244,-176.999,6.938,148.411
C07848=1201.178,261.373,-64.271,-176.997,6.940,148.411
C07849=1201.174,261.621,-64.299,-176.994,6.942,148.410
C07850=1201.170,261.871,-64.326,-176.992,6.945,148.410
C07851=1201.165,262.118,-64.354,-176.989,6.947,148.410
C07852=1201.161,262.367,-64.381,-176.986,6.950,148.410
C07853=1201.156,262.640,-64.412,-176.984,6.952,148.410
C07854=1201.151,262.913,-64.441,-176.981,6.955,148.410
C07855=1201.146,263.185,-64.472,-176.978,6.958,148.409
C07856=1201.141,263.458,-64.502,-176.975,6.961,148.409
C07857=1201.137,263.707,-64.529,-176.973,6.962,148.409
C07858=1201.132,263.955,-64.557,-176.970,6.965,148.409
C07859=1201.128,264.203,-64.584,-176.968,6.968,148.409
C07860=1201.124,264.453,-64.612,-176.965,6.969,148.409
C07861=1201.119,264.700,-64.639,-176.962,6.972,148.408
C07862=1201.115,264.949,-64.666,-176.960,6.975,148.408
C07863=1201.111,265.197,-64.695,-176.958,6.976,148.408
C07864=1201.106,265.446,-64.722,-176.955,6.979,148.408
C07865=1201.102,265.694,-64.749,-176.952,6.981,148.408
C07866=1201.097,265.942,-64.776,-176.950,6.984,148.408
C07867=1201.093,266.191,-64.805,-176.947,6.987,148.408
C07868=1201.088,266.439,-64.833,-176.944,6.989,148.407
C07869=1201.084,266.688,-64.860,-176.942,6.991,148.407
C07870=1201.080,266.936,-64.888,-176.940,6.994,148.407
C07871=1201.075,267.185,-64.915,-176.937,6.996,148.407
C07872=1201.071,267.433,-64.943,-176.935,6.998,148.407
C07873=1201.066,267.682,-64.971,-176.932,7.001,148.407
C07874=1201.062,267.930,-64.999,-176.929,7.003,148.407
C07875=1201.058,268.179,-65.027,-176.927,7.006,148.406
C07876=1201.053,268.427,-65.054,-176.924,7.008,148.406
C07877=1201.049,268.675,-65.082,-176.922,7.010,148.406
C07878=1201.045,268.924,-65.110,-176.919,7.013,148.406
C07879=1201.040,269.172,-65.138,-176.916,7.015,148.406
C07880=1201.036,269.420,-65.165,-176.914,7.018,148.406
C07881=1201.032,269.669,-65.193,-176.912,7.020,148.406
C07882=1201.027,269.917,-65.222,-176.908,7.023,148.405
C07883=1201.023,270.166,-65.249,-176.906,7.025,148.405
C07884=1201.018,270.414,-65.277,-176.904,7.028,148.405
C07885=1201.014,270.662,-65.305,-176.901,7.030,148.405
C07886=1201.010,270.911,-65.334,-176.899,7.032,148.405
C07887=1201.005,271.159,-65.361,-176.896,7.035,148.405
C07888=1201.001,271.408,-65.389,-176.894,7.037,148.405
C07889=1200.996,271.656,-65.417,-176.891,7.040,148.405
C07890=1200.992,271.905,-65.445,-176.889,7.042,148.404
C07891=1200.988,272.152,-65.473,-176.886,7.045,148.404
C07892=1200.983,272.401,-65.501,-176.883,7.047,148.404
C07893=1200.979,272.650,-65.529,-176.881,7.050,148.404
C07894=1200.974,272.898,-65.557,-176.879,7.052,148.404
C07895=1200.970,273.147,-65.585,-176.875,7.055,148.404
C07896=1200.966,273.394,-65.613,-176.873,7.057,148.404
C07897=1200.962,273.643,-65.641,-176.870,7.060,148.404
C07898=1200.957,273.891,-65.670,-176.868,7.062,148.404
C07899=1200.953,274.140,-65.698,-176.865,7.065,148.403
C07900=1200.949,274.388,-65.726,-176.863,7.067,148.403
C07901=1200.944,274.637,-65.754,-176.860,7.070,148.403
C07902=1200.940,274.884,-65.782,-176.858,7.072,148.403
C07903=1200.935,275.134,-65.810,-176.855,7.075,148.403
C07904=1200.931,275.382,-65.838,-176.853,7.077,148.403
C07905=1200.927,275.630,-65.866,-176.850,7.080,148.403
C07906=1200.922,275.879,-65.894,-176.848,7.082,148.402
C07907=1200.918,276.127,-65.923,-176.845,7.084,148.402
C07908=1200.913,276.375,-65.952,-176.843,7.087,148.402
C07909=1200.910,276.623,-65.980,-176.841,7.090,148.402
C07910=1200.904,276.871,-66.008,-176.837,7.092,148.402
C07911=1200.901,277.120,-66.036,-176.835,7.095,148.402
C07912=1200.896,277.368,-66.065,-176.833,7.098,148.402
C07913=1200.892,277.617,-66.093,-176.830,7.100,148.402
C07914=1200.887,277.866,-66.122,-176.827,7.102,148.402
C07915=1200.883,278.114,-66.149,-176.825,7.105,148.401
C07916=1200.879,278.362,-66.178,-176.822,7.108,148.401
C07917=1200.874,278.610,-66.206,-176.820,7.110,148.401
C07918=1200.870,278.859,-66.235,-176.817,7.112,148.401
C07919=1200.866,279.106,-66.263,-176.814,7.116,148.401
C07920=1200.861,279.355,-66.292,-176.812,7.118,148.401
C07921=1200.857,279.604,-66.320,-176.810,7.121,148.401
C07922=1200.852,279.852,-66.348,-176.807,7.123,148.401
C07923=1200.849,280.100,-66.377,-176.804,7.126,148.401
C07924=1200.844,280.348,-66.406,-176.802,7.128,148.401
C07925=1200.839,280.597,-66.434,-176.799,7.131,148.401
C07926=1200.836,280.846,-66.462,-176.797,7.133,148.400
C07927=1200.831,281.093,-66.492,-176.794,7.136,148.400
C07928=1200.827,281.342,-66.520,-176.792,7.138,148.400
C07929=1200.822,281.590,-66.548,-176.789,7.141,148.400
C07930=1200.818,281.838,-66.577,-176.787,7.143,148.400
C07931=1200.814,282.087,-66.606,-176.784,7.146,148.400
C07932=1200.809,282.335,-66.634,-176.782,7.148,148.400
C07933=1200.804,282.584,-66.663,-176.779,7.151,148.400
C07934=1200.801,282.832,-66.692,-176.777,7.153,148.400
C07935=1200.796,283.080,-66.720,-176.774,7.156,148.400
C07936=1200.792,283.328,-66.749,-176.772,7.158,148.400
C07937=1200.788,283.577,-66.778,-176.769,7.161,148.399
C07938=1200.783,283.825,-66.806,-176.766,7.164,148.399
C07939=1200.779,284.073,-66.835,-176.764,7.166,148.399
C07940=1200.775,284.322,-66.864,-176.761,7.169,148.399
C07941=1200.770,284.570,-66.893,-176.759,7.171,148.399
C07942=1200.766,284.818,-66.921,-176.756,7.174,148.399
C07943=1200.761,285.067,-66.951,-176.754,7.176,148.399
C07944=1200.757,285.315,-66.979,-176.751,7.179,148.399
C07945=1200.753,285.563,-67.008,-176.749,7.181,148.399
C07946=1200.748,285.812,-67.037,-176.746,7.184,148.399
C07947=1200.744,286.059,-67.066,-176.744,7.187,148.399
C07948=1200.740,286.308,-67.094,-176.741,7.189,148.398
C07949=1200.736,286.556,-67.123,-176.738,7.192,148.398
C07950=1200.731,286.805,-67.152,-176.736,7.195,148.398
C07951=1200.726,287.053,-67.181,-176.734,7.198,148.398
C07952=1200.722,287.302,-67.210,-176.731,7.200,148.398
C07953=1200.719,287.549,-67.239,-176.729,7.203,148.398
C07954=1200.714,287.798,-67.268,-176.727,7.205,148.398
C07955=1200.709,288.046,-67.297,-176.723,7.208,148.398
C07956=1200.705,288.294,-67.326,-176.721,7.211,148.398
C07957=1200.700,288.569,-67.358,-176.719,7.213,148.398
C07958=1200.696,288.843,-67.389,-176.716,7.216,148.398
C07959=1200.691,289.118,-67.423,-176.713,7.219,148.398
C07960=1200.686,289.392,-67.454,-176.710,7.222,148.397
C07961=1200.682,289.640,-67.484,-176.707,7.225,148.397
C07962=1200.677,289.888,-67.512,-176.705,7.227,148.397
C07963=1200.673,290.137,-67.542,-176.702,7.230,148.397
C07964=1200.669,290.385,-67.571,-176.700,7.233,148.397
C07965=1200.665,290.633,-67.600,-176.698,7.235,148.397
C07966=1200.660,290.882,-67.629,-176.695,7.238,148.397
C07967=1200.656,291.129,-67.658,-176.693,7.240,148.397
C07968=1200.652,291.378,-67.687,-176.690,7.243,148.397
C07969=1200.647,291.626,-67.717,-176.687,7.246,148.397
C07970=1200.643,291.874,-67.746,-176.685,7.248,148.397
C07971=1200.639,292.123,-67.775,-176.682,7.251,148.397
C07972=1200.635,292.371,-67.804,-176.680,7.253,148.397
C07973=1200.630,292.619,-67.833,-176.677,7.256,148.397
C07974=1200.626,292.867,-67.863,-176.675,7.259,148.397
C07975=1200.621,293.115,-67.892,-176.672,7.262,148.397
C07976=1200.617,293.364,-67.922,-176.670,7.265,148.397
C07977=1200.613,293.612,-67.951,-176.668,7.267,148.396
C07978=1200.609,293.861,-67.980,-176.665,7.270,148.396
C07979=1200.604,294.108,-68.009,-176.662,7.273,148.396
C07980=1200.600,294.357,-68.039,-176.660,7.275,148.396
C07981=1200.595,294.605,-68.068,-176.657,7.278,148.396
C07982=1200.591,294.853,-68.097,-176.655,7.280,148.396
C07983=1200.587,295.102,-68.127,-176.652,7.283,148.396
C07984=1200.583,295.350,-68.156,-176.649,7.286,148.396
C07985=1200.579,295.598,-68.186,-176.647,7.288,148.396
C07986=1200.574,295.846,-68.215,-176.645,7.291,148.396
C07987=1200.570,296.095,-68.245,-176.642,7.293,148.396
C07988=1200.566,296.343,-68.274,-176.640,7.296,148.396
C07989=1200.561,296.591,-68.304,-176.637,7.299,148.396
C07990=1200.556,296.839,-68.333,-176.635,7.302,148.396
C07991=1200.552,297.087,-68.363,-176.632,7.305,148.396
C07992=1200.548,297.336,-68.392,-176.630,7.307,148.396
C07993=1200.544,297.584,-68.422,-176.627,7.310,148.396
C07994=1200.540,297.831,-68.452,-176.625,7.313,148.396
C07995=1200.536,298.080,-68.481,-176.622,7.315,148.396
C07996=1200.532,298.328,-68.511,-176.620,7.318,148.396
C07997=1200.527,298.577,-68.541,-176.617,7.321,148.396
C07998=1200.523,298.825,-68.570,-176.615,7.323,148.395
C07999=1200.518,299.073,-68.600,-176.612,7.326,148.395
C08000=1200.514,299.321,-68.629,-176.610,7.328,148.395
C08001=1200.510,299.569,-68.659,-176.607,7.331,148.395
C08002=1200.505,299.818,-68.689,-176.605,7.334,148.395
C08003=1200.501,300.066,-68.719,-176.603,7.337,148.395
C08004=1200.497,300.314,-68.748,-176.600,7.340,148.395
C08005=1200.493,300.562,-68.778,-176.597,7.343,148.395
C08006=1200.488,300.810,-68.809,-176.595,7.345,148.395
C08007=1200.484,301.059,-68.838,-176.592,7.348,148.395
C08008=1200.480,301.307,-68.867,-176.590,7.350,148.395
C08009=1200.476,301.555,-68.898,-176.588,7.353,148.395
C08010=1200.471,301.803,-68.928,-176.585,7.356,148.395
C08011=1200.467,302.051,-68.957,-176.583,7.358,148.395
C08012=1200.463,302.300,-68.987,-176.580,7.361,148.395
C08013=1200.459,302.547,-69.017,-176.577,7.364,148.395
C08014=1200.454,302.796,-69.047,-176.576,7.367,148.395
C08015=1200.450,303.044,-69.077,-176.573,7.370,148.395
C08016=1200.446,303.292,-69.106,-176.570,7.373,148.395
C08017=1200.441,303.540,-69.136,-176.568,7.375,148.395
C08018=1200.437,303.788,-69.167,-176.565,7.378,148.395
C08019=1200.433,304.036,-69.196,-176.563,7.381,148.395
C08020=1200.428,304.284,-69.227,-176.561,7.383,148.395
C08021=1200.424,304.533,-69.256,-176.558,7.386,148.395
C08022=1200.419,304.781,-69.286,-176.555,7.389,148.395
C08023=1200.415,305.029,-69.316,-176.553,7.391,148.395
C08024=1200.412,305.278,-69.346,-176.550,7.395,148.395
C08025=1200.407,305.526,-69.377,-176.548,7.397,148.395
C08026=1200.403,305.774,-69.407,-176.546,7.400,148.395
C08027=1200.398,306.022,-69.437,-176.543,7.403,148.395
C08028=1200.394,306.270,-69.467,-176.541,7.405,148.395
C08029=1200.390,306.518,-69.497,-176.539,7.408,148.395
C08030=1200.385,306.766,-69.527,-176.536,7.411,148.395
C08031=1200.381,307.014,-69.557,-176.534,7.413,148.395
C08032=1200.377,307.262,-69.588,-176.531,7.417,148.395
C08033=1200.373,307.510,-69.617,-176.528,7.420,148.395
C08034=1200.369,307.759,-69.648,-176.526,7.422,148.395
C08035=1200.364,308.007,-69.678,-176.524,7.425,148.395
C08036=1200.360,308.255,-69.709,-176.521,7.428,148.395
C08037=1200.356,308.503,-69.739,-176.519,7.430,148.395
C08038=1200.351,308.751,-69.769,-176.516,7.433,148.395
C08039=1200.347,308.999,-69.799,-176.514,7.436,148.395
C08040=1200.343,309.247,-69.830,-176.512,7.438,148.395
C08041=1200.339,309.496,-69.860,-176.509,7.442,148.395
C08042=1200.334,309.744,-69.890,-176.507,7.445,148.395
C08043=1200.330,309.992,-69.921,-176.505,7.447,148.395
C08044=1200.326,310.240,-69.951,-176.502,7.450,148.395
C08045=1200.322,310.488,-69.981,-176.499,7.453,148.395
C08046=1200.317,310.736,-70.012,-176.497,7.455,148.395
C08047=1200.314,310.984,-70.042,-176.494,7.458,148.395
C08048=1200.309,311.233,-70.072,-176.492,7.462,148.395
C08049=1200.304,311.481,-70.103,-176.490,7.464,148.395
C08050=1200.300,311.728,-70.133,-176.487,7.467,148.395
C08051=1200.296,311.976,-70.164,-176.485,7.470,148.395
C08052=1200.292,312.225,-70.194,-176.482,7.473,148.395
C08053=1200.288,312.473,-70.224,-176.480,7.475,148.395
C08054=1200.283,312.721,-70.255,-176.478,7.478,148.395
C08055=1200.279,312.969,-70.285,-176.475,7.481,148.395
C08056=1200.275,313.217,-70.316,-176.473,7.484,148.395
C08057=1200.270,313.465,-70.347,-176.471,7.487,148.395
C08058=1200.267,313.713,-70.377,-176.468,7.490,148.395
C08059=1200.262,313.961,-70.408,-176.466,7.492,148.395
C08060=1200.258,314.210,-70.439,-176.463,7.495,148.395
C08061=1200.253,314.486,-70.473,-176.460,7.498,148.395
C08062=1200.248,314.762,-70.507,-176.458,7.502,148.395
C08063=1200.244,315.039,-70.541,-176.455,7.505,148.395
C08064=1200.239,315.315,-70.575,-176.453,7.508,148.395
C08065=1200.235,315.562,-70.606,-176.450,7.511,148.395
C08066=1200.230,315.810,-70.636,-176.447,7.514,148.395
C08067=1200.226,316.059,-70.667,-176.446,7.516,148.396
C08068=1200.222,316.307,-70.698,-176.443,7.519,148.396
C08069=1200.218,316.555,-70.728,-176.440,7.522,148.396
C08070=1200.214,316.803,-70.759,-176.438,7.525,148.396
C08071=1200.209,317.051,-70.790,-176.436,7.528,148.396
C08072=1200.205,317.299,-70.821,-176.433,7.531,148.396
C08073=1200.201,317.548,-70.852,-176.431,7.534,148.396
C08074=1200.197,317.795,-70.883,-176.429,7.536,148.396
C08075=1200.192,318.043,-70.914,-176.426,7.539,148.396
C08076=1200.188,318.292,-70.945,-176.423,7.542,148.396
C08077=1200.184,318.539,-70.976,-176.422,7.545,148.396
C08078=1200.180,318.787,-71.006,-176.419,7.548,148.396
C08079=1200.176,319.036,-71.037,-176.416,7.551,148.396
C08080=1200.171,319.284,-71.068,-176.414,7.554,148.396
C08081=1200.167,319.531,-71.099,-176.412,7.556,148.396
C08082=1200.163,319.780,-71.130,-176.409,7.559,148.396
C08083=1200.158,320.028,-71.161,-176.407,7.563,148.396
C08084=1200.155,320.276,-71.192,-176.405,7.565,148.396
C08085=1200.150,320.524,-71.222,-176.402,7.568,148.396
C08086=1200.146,320.771,-71.254,-176.400,7.571,148.397
C08087=1200.142,321.020,-71.285,-176.398,7.574,148.396
C08088=1200.138,321.268,-71.316,-176.395,7.577,148.396
C08089=1200.133,321.515,-71.347,-176.393,7.580,148.397
C08090=1200.129,321.764,-71.378,-176.390,7.583,148.397
C08091=1200.125,322.012,-71.409,-176.389,7.585,148.397
C08092=1200.121,322.261,-71.440,-176.386,7.588,148.397
C08093=1200.116,322.508,-71.472,-176.383,7.591,148.397
C08094=1200.113,322.756,-71.502,-176.382,7.594,148.397
C08095=1200.109,323.004,-71.534,-176.379,7.597,148.397
C08096=1200.104,323.252,-71.565,-176.377,7.600,148.397
C08097=1200.100,323.500,-71.596,-176.375,7.603,148.397
C08098=1200.096,323.748,-71.627,-176.372,7.606,148.397
C08099=1200.092,323.996,-71.658,-176.370,7.609,148.397
C08100=1200.087,324.244,-71.690,-176.367,7.612,148.397
C08101=1200.083,324.492,-71.721,-176.365,7.614,148.398
C08102=1200.079,324.740,-71.752,-176.363,7.617,148.398
C08103=1200.075,324.988,-71.784,-176.360,7.621,148.398
C08104=1200.070,325.236,-71.814,-176.358,7.623,148.398
C08105=1200.067,325.484,-71.846,-176.356,7.626,148.398
C08106=1200.062,325.732,-71.877,-176.353,7.629,148.398
C08107=1200.058,325.980,-71.909,-176.351,7.632,148.398
C08108=1200.054,326.228,-71.940,-176.349,7.635,148.398
C08109=1200.050,326.476,-71.971,-176.346,7.638,148.398
C08110=1200.046,326.724,-72.002,-176.344,7.641,148.398
C08111=1200.041,326.973,-72.035,-176.342,7.643,148.398
C08112=1200.037,327.220,-72.066,-176.340,7.647,148.398
C08113=1200.033,327.469,-72.097,-176.337,7.650,148.398
C08114=1200.028,327.716,-72.129,-176.335,7.653,148.399
C08115=1200.024,327.965,-72.160,-176.333,7.655,148.399
C08116=1200.020,328.212,-72.191,-176.331,7.659,148.399
C08117=1200.016,328.460,-72.223,-176.328,7.662,148.399
C08118=1200.012,328.708,-72.254,-176.326,7.664,148.399
C08119=1200.008,328.956,-72.286,-176.323,7.667,148.399
C08120=1200.003,329.204,-72.318,-176.321,7.671,148.399
C08121=1199.999,329.452,-72.349,-176.319,7.674,148.399
C08122=1199.995,329.700,-72.380,-176.317,7.676,148.399
C08123=1199.991,329.948,-72.412,-176.315,7.679,148.400
C08124=1199.986,330.196,-72.443,-176.312,7.682,148.400
C08125=1199.982,330.444,-72.475,-176.310,7.685,148.400
C08126=1199.978,330.692,-72.507,-176.308,7.688,148.400
C08127=1199.974,330.939,-72.539,-176.305,7.691,148.400
C08128=1199.970,331.188,-72.570,-176.303,7.694,148.400
C08129=1199.966,331.435,-72.601,-176.301,7.697,148.400
C08130=1199.961,331.684,-72.634,-176.299,7.700,148.400
C08131=1199.957,331.932,-72.666,-176.296,7.703,148.400
C08132=1199.953,332.179,-72.697,-176.294,7.706,148.401
C08133=1199.949,332.428,-72.728,-176.292,7.709,148.401
C08134=1199.944,332.675,-72.760,-176.290,7.712,148.401
C08135=1199.940,332.923,-72.792,-176.287,7.715,148.401
C08136=1199.937,333.171,-72.824,-176.285,7.718,148.401
C08137=1199.932,333.419,-72.856,-176.283,7.721,148.401
C08138=1199.928,333.667,-72.888,-176.281,7.724,148.401
C08139=1199.924,333.914,-72.919,-176.278,7.727,148.401
C08140=1199.920,334.162,-72.951,-176.276,7.730,148.402
C08141=1199.916,334.411,-72.984,-176.274,7.733,148.402
C08142=1199.911,334.658,-73.015,-176.271,7.736,148.402
C08143=1199.907,334.907,-73.046,-176.270,7.739,148.402
C08144=1199.903,335.155,-73.079,-176.268,7.742,148.402
C08145=1199.898,335.402,-73.110,-176.265,7.745,148.402
C08146=1199.895,335.650,-73.142,-176.263,7.748,148.402
C08147=1199.890,335.899,-73.175,-176.261,7.751,148.403
C08148=1199.886,336.146,-73.206,-176.259,7.754,148.403
C08149=1199.882,336.394,-73.238,-176.256,7.757,148.403
C08150=1199.878,336.643,-73.270,-176.254,7.760,148.403
C08151=1199.874,336.889,-73.302,-176.252,7.763,148.403
C08152=1199.869,337.138,-73.335,-176.250,7.766,148.403
C08153=1199.866,337.386,-73.367,-176.247,7.769,148.403
C08154=1199.862,337.634,-73.399,-176.246,7.772,148.404
C08155=1199.857,337.881,-73.431,-176.243,7.775,148.404
C08156=1199.853,338.129,-73.463,-176.241,7.778,148.404
C08157=1199.849,338.378,-73.495,-176.239,7.781,148.404
C08158=1199.844,338.625,-73.526,-176.237,7.784,148.404
C08159=1199.840,338.873,-73.559,-176.235,7.787,148.404
C08160=1199.837,339.121,-73.591,-176.232,7.791,148.405
C08161=1199.833,339.369,-73.623,-176.230,7.793,148.405
C08162=1199.828,339.617,-73.655,-176.228,7.796,148.405
C08163=1199.824,339.865,-73.687,-176.226,7.800,148.405
C08164=1199.820,340.113,-73.720,-176.224,7.802,148.405
C08165=1199.815,340.391,-73.756,-176.221,7.806,148.405
C08166=1199.810,340.669,-73.792,-176.219,7.809,148.406
C08167=1199.806,340.948,-73.829,-176.216,7.813,148.406
C08168=1199.800,341.226,-73.864,-176.214,7.816,148.406
C08169=1199.797,341.474,-73.897,-176.212,7.819,148.406
C08170=1199.793,341.722,-73.929,-176.210,7.823,148.406
C08171=1199.789,341.970,-73.961,-176.208,7.825,148.407
C08172=1199.784,342.217,-73.994,-176.206,7.829,148.407
C08173=1199.780,342.465,-74.026,-176.203,7.832,148.407
C08174=1199.776,342.714,-74.058,-176.201,7.834,148.407
C08175=1199.773,342.961,-74.091,-176.199,7.837,148.407
C08176=1199.768,343.209,-74.123,-176.197,7.841,148.407
C08177=1199.763,343.457,-74.155,-176.195,7.844,148.408
C08178=1199.760,343.704,-74.188,-176.193,7.847,148.408
C08179=1199.755,343.953,-74.220,-176.191,7.850,148.408
C08180=1199.751,344.201,-74.253,-176.189,7.853,148.408
C08181=1199.747,344.449,-74.285,-176.187,7.856,148.408
C08182=1199.742,344.696,-74.318,-176.185,7.859,148.409
C08183=1199.739,344.944,-74.350,-176.183,7.862,148.409
C08184=1199.734,345.192,-74.383,-176.181,7.865,148.409
C08185=1199.730,345.440,-74.416,-176.179,7.868,148.409
C08186=1199.727,345.688,-74.448,-176.176,7.872,148.409
C08187=1199.722,345.935,-74.481,-176.174,7.875,148.410
C08188=1199.718,346.184,-74.513,-176.173,7.877,148.410
C08189=1199.713,346.431,-74.546,-176.170,7.881,148.410
C08190=1199.710,346.679,-74.578,-176.168,7.884,148.410
C08191=1199.705,346.927,-74.611,-176.166,7.887,148.411
C08192=1199.701,347.175,-74.643,-176.164,7.890,148.411
C08193=1199.698,347.422,-74.676,-176.162,7.893,148.411
C08194=1199.693,347.671,-74.708,-176.160,7.897,148.411
C08195=1199.689,347.918,-74.742,-176.158,7.899,148.411
C08196=1199.685,348.166,-74.775,-176.156,7.902,148.412
C08197=1199.681,348.413,-74.806,-176.154,7.906,148.412
C08198=1199.676,348.661,-74.839,-176.152,7.908,148.412
C08199=1199.672,348.910,-74.872,-176.150,7.912,148.412
C08200=1199.668,349.157,-74.905,-176.148,7.915,148.412
C08201=1199.664,349.405,-74.938,-176.146,7.918,148.413
C08202=1199.660,349.653,-74.970,-176.144,7.921,148.413
C08203=1199.656,349.901,-75.003,-176.142,7.924,148.413
C08204=1199.652,350.149,-75.036,-176.140,7.928,148.413
C08205=1199.647,350.397,-75.069,-176.138,7.930,148.414
C08206=1199.644,350.644,-75.101,-176.136,7.934,148.414
C08207=1199.640,350.892,-75.134,-176.133,7.937,148.414
C08208=1199.636,351.140,-75.168,-176.132,7.940,148.414
C08209=1199.631,351.387,-75.200,-176.130,7.943,148.415
C08210=1199.626,351.635,-75.233,-176.128,7.946,148.415
C08211=1199.622,351.883,-75.266,-176.126,7.949,148.415
C08212=1199.619,352.130,-75.299,-176.124,7.952,148.415
C08213=1199.614,352.379,-75.331,-176.122,7.956,148.416
C08214=1199.610,352.626,-75.364,-176.120,7.958,148.416
C08215=1199.606,352.874,-75.397,-176.118,7.962,148.416
C08216=1199.602,353.122,-75.430,-176.116,7.965,148.416
C08217=1199.598,353.370,-75.464,-176.114,7.969,148.417
C08218=1199.594,353.617,-75.497,-176.113,7.971,148.417
C08219=1199.589,353.866,-75.529,-176.110,7.975,148.417
C08220=1199.585,354.113,-75.562,-176.108,7.978,148.417
C08221=1199.581,354.361,-75.595,-176.107,7.981,148.418
C08222=1199.578,354.609,-75.628,-176.105,7.984,148.418
C08223=1199.574,354.856,-75.661,-176.102,7.987,148.418
C08224=1199.569,355.104,-75.694,-176.101,7.990,148.419
C08225=1199.565,355.352,-75.728,-176.099,7.994,148.419
C08226=1199.561,355.599,-75.761,-176.097,7.997,148.419
C08227=1199.557,355.847,-75.794,-176.096,8.000,148.420
C08228=1199.553,356.095,-75.827,-176.093,8.003,148.420
C08229=1199.549,356.343,-75.860,-176.091,8.006,148.420
C08230=1199.545,356.590,-75.893,-176.090,8.009,148.420
C08231=1199.541,356.839,-75.927,-176.088,8.013,148.421
C08232=1199.537,357.087,-75.960,-176.085,8.016,148.421
C08233=1199.533,357.334,-75.993,-176.084,8.019,148.421
C08234=1199.529,357.582,-76.026,-176.082,8.022,148.421
C08235=1199.524,357.830,-76.059,-176.080,8.026,148.422
C08236=1199.520,358.077,-76.093,-176.079,8.028,148.422
C08237=1199.516,358.325,-76.126,-176.077,8.032,148.423
C08238=1199.512,358.573,-76.159,-176.075,8.035,148.423
C08239=1199.508,358.821,-76.192,-176.073,8.038,148.423
C08240=1199.504,359.068,-76.225,-176.071,8.041,148.423
C08241=1199.500,359.315,-76.259,-176.069,8.045,148.424
C08242=1199.495,359.563,-76.293,-176.068,8.047,148.424
C08243=1199.491,359.811,-76.326,-176.065,8.051,148.424
C08244=1199.487,360.060,-76.360,-176.064,8.054,148.425
C08245=1199.483,360.307,-76.393,-176.062,8.057,148.425
C08246=1199.479,360.555,-76.426,-176.060,8.061,148.425
C08247=1199.475,360.802,-76.460,-176.059,8.063,148.426
C08248=1199.471,361.050,-76.493,-176.057,8.067,148.426
C08249=1199.467,361.298,-76.526,-176.055,8.070,148.426
C08250=1199.463,361.545,-76.559,-176.053,8.073,148.426
C08251=1199.459,361.793,-76.592,-176.052,8.076,148.427
C08252=1199.455,362.041,-76.627,-176.050,8.080,148.427
C08253=1199.451,362.289,-76.660,-176.048,8.083,148.428
C08254=1199.446,362.537,-76.693,-176.046,8.086,148.428
C08255=1199.442,362.784,-76.727,-176.045,8.089,148.428
C08256=1199.439,363.032,-76.760,-176.043,8.092,148.429
C08257=1199.434,363.279,-76.794,-176.042,8.095,148.429
C08258=1199.430,363.528,-76.828,-176.040,8.099,148.429
C08259=1199.426,363.775,-76.862,-176.038,8.102,148.430
C08260=1199.422,364.023,-76.895,-176.036,8.105,148.430
C08261=1199.418,364.271,-76.928,-176.035,8.109,148.430
C08262=1199.414,364.518,-76.962,-176.033,8.111,148.431
C08263=1199.409,364.766,-76.996,-176.031,8.115,148.431
C08264=1199.406,365.014,-77.030,-176.030,8.118,148.431
C08265=1199.402,365.261,-77.063,-176.028,8.121,148.432
C08266=1199.398,365.509,-77.096,-176.027,8.124,148.432
C08267=1199.394,365.756,-77.130,-176.025,8.127,148.433
C08268=1199.390,366.005,-77.164,-176.024,8.130,148.433
C08269=1199.386,366.285,-77.202,-176.022,8.134,148.433
C08270=1199.381,366.566,-77.241,-176.020,8.137,148.434
C08271=1199.376,366.847,-77.278,-176.018,8.141,148.434
C08272=1199.371,367.128,-77.317,-176.016,8.145,148.435
C08273=1199.367,367.375,-77.351,-176.015,8.148,148.435
C08274=1199.363,367.622,-77.384,-176.013,8.151,148.436
C08275=1199.359,367.870,-77.418,-176.012,8.155,148.436
C08276=1199.355,368.118,-77.452,-176.010,8.158,148.436
C08277=1199.351,368.365,-77.486,-176.009,8.161,148.437
C08278=1199.346,368.613,-77.519,-176.008,8.164,148.437
C08279=1199.343,368.861,-77.553,-176.006,8.167,148.438
C08280=1199.339,369.109,-77.587,-176.005,8.170,148.438
C08281=1199.334,369.356,-77.621,-176.003,8.173,148.438
C08282=1199.331,369.604,-77.655,-176.002,8.177,148.439
C08283=1199.326,369.851,-77.688,-176.000,8.180,148.439
C08284=1199.322,370.099,-77.723,-175.999,8.182,148.440
C08285=1199.318,370.347,-77.756,-175.997,8.186,148.440
C08286=1199.314,370.595,-77.791,-175.996,8.189,148.440
C08287=1199.311,370.842,-77.825,-175.994,8.193,148.441
C08288=1199.306,371.090,-77.858,-175.993,8.195,148.441
C08289=1199.302,371.337,-77.893,-175.992,8.198,148.442
C08290=1199.298,371.585,-77.926,-175.990,8.202,148.442
C08291=1199.294,371.833,-77.960,-175.989,8.205,148.442
C08292=1199.290,372.080,-77.994,-175.988,8.207,148.443
C08293=1199.286,372.328,-78.028,-175.986,8.211,148.443
C08294=1199.282,372.576,-78.062,-175.985,8.214,148.444
C08295=1199.278,372.823,-78.096,-175.984,8.217,148.444
C08296=1199.273,373.071,-78.131,-175.982,8.221,148.445
C08297=1199.270,373.319,-78.164,-175.981,8.223,148.445
C08298=1199.266,373.566,-78.198,-175.980,8.226,148.445
C08299=1199.261,373.814,-78.233,-175.978,8.230,148.446
C08300=1199.258,374.061,-78.267,-175.977,8.233,148.447
C08301=1199.253,374.310,-78.301,-175.976,8.236,148.447
C08302=1199.250,374.557,-78.335,-175.975,8.239,148.447
C08303=1199.245,374.804,-78.369,-175.973,8.242,148.448
C08304=1199.242,375.052,-78.403,-175.972,8.245,148.448
C08305=1199.237,375.300,-78.437,-175.971,8.248,148.449
C08306=1199.234,375.548,-78.471,-175.970,8.251,148.449
C08307=1199.229,375.795,-78.506,-175.968,8.255,148.450
C08308=1199.225,376.042,-78.540,-175.967,8.258,148.450
C08309=1199.221,376.290,-78.574,-175.966,8.260,148.451
C08310=1199.217,376.538,-78.608,-175.965,8.263,148.451
C08311=1199.213,376.786,-78.642,-175.964,8.266,148.451
C08312=1199.209,377.033,-78.676,-175.962,8.270,148.452
C08313=1199.205,377.281,-78.711,-175.961,8.273,148.452
C08314=1199.201,377.528,-78.745,-175.960,8.276,148.453
C08315=1199.197,377.776,-78.779,-175.959,8.279,148.453
C08316=1199.192,378.023,-78.814,-175.958,8.282,148.454
C08317=1199.189,378.271,-78.848,-175.957,8.285,148.454
C08318=1199.185,378.519,-78.883,-175.956,8.287,148.455
C08319=1199.181,378.766,-78.916,-175.954,8.291,148.455
C08320=1199.177,379.014,-78.951,-175.953,8.294,148.456
C08321=1199.173,379.261,-78.985,-175.952,8.297,148.456
C08322=1199.168,379.509,-79.019,-175.951,8.300,148.457
C08323=1199.164,379.757,-79.054,-175.950,8.303,148.457
C08324=1199.160,380.004,-79.088,-175.949,8.306,148.458
C08325=1199.156,380.252,-79.122,-175.948,8.309,148.458
C08326=1199.152,380.500,-79.157,-175.947,8.312,148.459
C08327=1199.148,380.748,-79.191,-175.946,8.315,148.459
C08328=1199.144,380.995,-79.226,-175.945,8.318,148.460
C08329=1199.140,381.242,-79.259,-175.944,8.321,148.460
C08330=1199.136,381.490,-79.294,-175.943,8.324,148.461
C08331=1199.132,381.738,-79.329,-175.942,8.327,148.461
C08332=1199.128,381.986,-79.363,-175.942,8.330,148.462
C08333=1199.124,382.232,-79.398,-175.940,8.333,148.462
C08334=1199.119,382.480,-79.433,-175.940,8.336,148.463
C08335=1199.116,382.728,-79.467,-175.938,8.339,148.463
C08336=1199.112,382.975,-79.501,-175.938,8.342,148.464
C08337=1199.108,383.223,-79.536,-175.937,8.345,148.464
C08338=1199.104,383.470,-79.570,-175.936,8.348,148.465
C08339=1199.100,383.718,-79.605,-175.935,8.351,148.465
C08340=1199.095,383.966,-79.639,-175.934,8.354,148.466
C08341=1199.092,384.214,-79.674,-175.933,8.357,148.466
C08342=1199.088,384.461,-79.708,-175.932,8.360,148.467
C08343=1199.084,384.709,-79.743,-175.932,8.362,148.467
C08344=1199.080,384.956,-79.777,-175.931,8.365,148.468
C08345=1199.075,385.203,-79.812,-175.930,8.368,148.468
C08346=1199.071,385.451,-79.847,-175.929,8.371,148.469
C08347=1199.067,385.699,-79.881,-175.928,8.374,148.469
C08348=1199.064,385.946,-79.915,-175.927,8.377,148.470
C08349=1199.059,386.194,-79.950,-175.927,8.379,148.470
C08350=1199.055,386.441,-79.986,-175.926,8.382,148.471
C08351=1199.051,386.689,-80.020,-175.925,8.385,148.471
C08352=1199.048,386.937,-80.054,-175.924,8.388,148.472
C08353=1199.043,387.184,-80.089,-175.923,8.391,148.473
C08354=1199.039,387.432,-80.124,-175.923,8.394,148.473
C08355=1199.035,387.679,-80.159,-175.922,8.397,148.474
C08356=1199.032,387.927,-80.193,-175.921,8.399,148.474
C08357=1199.027,388.174,-80.227,-175.921,8.402,148.475
C08358=1199.023,388.422,-80.262,-175.920,8.405,148.475
C08359=1199.019,388.669,-80.297,-175.919,8.408,148.476
C08360=1199.016,388.917,-80.332,-175.918,8.411,148.476
C08361=1199.011,389.164,-80.366,-175.918,8.413,148.477
C08362=1199.007,389.412,-80.401,-175.917,8.416,148.477
C08363=1199.003,389.659,-80.436,-175.916,8.419,148.478
C08364=1198.999,389.907,-80.471,-175.916,8.422,148.478
C08365=1198.995,390.154,-80.505,-175.915,8.425,148.479
C08366=1198.991,390.402,-80.540,-175.915,8.427,148.480
C08367=1198.987,390.650,-80.575,-175.914,8.430,148.480
C08368=1198.983,390.897,-80.610,-175.913,8.433,148.481
C08369=1198.979,391.145,-80.645,-175.913,8.435,148.481
C08370=1198.975,391.392,-80.679,-175.912,8.438,148.482
C08371=1198.971,391.640,-80.714,-175.912,8.440,148.482
C08372=1198.967,391.887,-80.749,-175.911,8.444,148.483
C08373=1198.962,392.170,-80.788,-175.910,8.447,148.483
C08374=1198.958,392.453,-80.829,-175.909,8.450,148.484
C08375=1198.953,392.736,-80.868,-175.909,8.453,148.485
C08376=1198.948,393.019,-80.909,-175.909,8.455,148.485
C08377=1198.944,393.267,-80.943,-175.908,8.458,148.486
C08378=1198.941,393.514,-80.977,-175.907,8.460,148.486
C08379=1198.937,393.762,-81.013,-175.907,8.464,148.487
C08380=1198.932,394.009,-81.047,-175.906,8.466,148.487
C08381=1198.929,394.257,-81.083,-175.906,8.469,148.488
C08382=1198.925,394.505,-81.118,-175.905,8.471,148.489
C08383=1198.921,394.752,-81.153,-175.905,8.474,148.489
C08384=1198.917,395.000,-81.188,-175.904,8.477,148.490
C08385=1198.913,395.247,-81.221,-175.903,8.480,148.490
C08386=1198.909,395.494,-81.257,-175.903,8.482,148.491
C08387=1198.904,395.742,-81.292,-175.903,8.484,148.491
C08388=1198.901,395.989,-81.327,-175.902,8.487,148.492
C08389=1198.897,396.237,-81.362,-175.902,8.490,148.492
C08390=1198.893,396.484,-81.397,-175.901,8.493,148.493
C08391=1198.889,396.732,-81.432,-175.901,8.495,148.494
C08392=1198.884,396.979,-81.467,-175.900,8.497,148.494
C08393=1198.880,397.227,-81.502,-175.900,8.500,148.494
C08394=1198.877,397.475,-81.537,-175.899,8.502,148.495
C08395=1198.872,397.722,-81.572,-175.899,8.505,148.496
C08396=1198.869,397.970,-81.607,-175.898,8.508,148.496
C08397=1198.865,398.217,-81.641,-175.898,8.510,148.497
C08398=1198.861,398.464,-81.677,-175.898,8.512,148.497
C08399=1198.856,398.712,-81.711,-175.898,8.514,148.498
C08400=1198.853,398.959,-81.747,-175.897,8.518,148.498
C08401=1198.849,399.207,-81.782,-175.897,8.520,148.499
C08402=1198.845,399.454,-81.817,-175.896,8.522,148.499
C08403=1198.841,399.702,-81.852,-175.896,8.524,148.500
C08404=1198.837,399.950,-81.887,-175.895,8.527,148.500
C08405=1198.832,400.197,-81.922,-175.895,8.530,148.501
C08406=1198.829,400.445,-81.957,-175.895,8.532,148.502
C08407=1198.824,400.692,-81.992,-175.895,8.534,148.502
C08408=1198.820,400.939,-82.027,-175.894,8.537,148.503
C08409=1198.817,401.187,-82.063,-175.894,8.540,148.503
C08410=1198.812,401.434,-82.097,-175.893,8.542,148.504
C08411=1198.809,401.682,-82.133,-175.893,8.544,148.504
C08412=1198.805,401.930,-82.168,-175.893,8.546,148.505
C08413=1198.800,402.177,-82.203,-175.892,8.550,148.505
C08414=1198.797,402.424,-82.238,-175.892,8.552,148.506
C08415=1198.792,402.672,-82.273,-175.892,8.554,148.506
C08416=1198.788,402.919,-82.308,-175.891,8.556,148.507
C08417=1198.784,403.167,-82.343,-175.891,8.558,148.507
C08418=1198.780,403.414,-82.378,-175.891,8.561,148.508
C08419=1198.777,403.662,-82.414,-175.890,8.563,148.508
C08420=1198.773,403.910,-82.449,-175.890,8.566,148.509
C08421=1198.768,404.157,-82.484,-175.889,8.568,148.509
C08422=1198.765,404.404,-82.520,-175.889,8.570,148.510
C08423=1198.761,404.652,-82.554,-175.889,8.573,148.511
C08424=1198.756,404.899,-82.590,-175.889,8.575,148.511
C08425=1198.753,405.146,-82.625,-175.888,8.577,148.512
C08426=1198.749,405.395,-82.660,-175.888,8.580,148.512
C08427=1198.745,405.641,-82.695,-175.888,8.582,148.513
C08428=1198.741,405.889,-82.731,-175.888,8.584,148.513
C08429=1198.737,406.137,-82.766,-175.887,8.586,148.514
C08430=1198.733,406.384,-82.801,-175.887,8.589,148.514
C08431=1198.729,406.631,-82.836,-175.887,8.591,148.515
C08432=1198.725,406.879,-82.871,-175.887,8.593,148.515
C08433=1198.721,407.126,-82.906,-175.887,8.595,148.516
C08434=1198.717,407.374,-82.942,-175.886,8.598,148.516
C08435=1198.712,407.622,-82.977,-175.886,8.600,148.517
C08436=1198.708,407.869,-83.012,-175.885,8.602,148.517
C08437=1198.704,408.116,-83.048,-175.885,8.604,148.518
C08438=1198.701,408.364,-83.084,-175.885,8.606,148.518
C08439=1198.696,408.611,-83.118,-175.885,8.609,148.519
C08440=1198.693,408.859,-83.154,-175.884,8.611,148.519
C08441=1198.689,409.106,-83.189,-175.884,8.613,148.520
C08442=1198.685,409.353,-83.224,-175.884,8.616,148.520
C08443=1198.681,409.601,-83.259,-175.884,8.618,148.521
C08444=1198.677,409.849,-83.295,-175.884,8.620,148.521
C08445=1198.673,410.096,-83.330,-175.883,8.622,148.522
C08446=1198.669,410.343,-83.365,-175.883,8.625,148.522
C08447=1198.665,410.591,-83.400,-175.882,8.627,148.523
C08448=1198.661,410.839,-83.436,-175.882,8.629,148.523
C08449=1198.656,411.086,-83.472,-175.882,8.631,148.524
C08450=1198.653,411.333,-83.507,-175.882,8.633,148.524
C08451=1198.649,411.581,-83.543,-175.881,8.636,148.525
C08452=1198.645,411.828,-83.577,-175.881,8.638,148.525
C08453=1198.641,412.076,-83.613,-175.881,8.640,148.526
C08454=1198.637,412.323,-83.648,-175.881,8.642,148.526
C08455=1198.633,412.570,-83.683,-175.881,8.644,148.527
C08456=1198.629,412.818,-83.720,-175.880,8.646,148.527
C08457=1198.625,413.066,-83.754,-175.880,8.648,148.528
C08458=1198.621,413.314,-83.790,-175.880,8.650,148.528
C08459=1198.617,413.560,-83.825,-175.880,8.653,148.529
C08460=1198.613,413.808,-83.861,-175.879,8.655,148.529
C08461=1198.609,414.055,-83.896,-175.879,8.657,148.530
C08462=1198.605,414.303,-83.931,-175.880,8.659,148.530
C08463=1198.601,414.550,-83.966,-175.879,8.661,148.531
C08464=1198.597,414.798,-84.002,-175.879,8.663,148.531
C08465=1198.593,415.046,-84.038,-175.878,8.665,148.532
C08466=1198.589,415.292,-84.073,-175.878,8.667,148.532
C08467=1198.585,415.540,-84.109,-175.878,8.670,148.533
C08468=1198.581,415.787,-84.144,-175.878,8.671,148.533
C08469=1198.576,416.117,-84.191,-175.877,8.674,148.534
C08470=1198.572,416.446,-84.238,-175.877,8.676,148.534
C08471=1198.571,416.776,-84.286,-175.877,8.680,148.535
C08472=1198.573,417.104,-84.331,-175.877,8.682,148.536
C08473=1198.152,417.105,-84.370,-175.880,8.693,148.539
C08474=1198.150,416.773,-84.324,-175.880,8.690,148.539
C08475=1198.150,416.441,-84.277,-175.880,8.687,148.538
C08476=1198.154,416.109,-84.229,-175.881,8.685,148.538
C08477=1198.159,415.777,-84.181,-175.881,8.681,148.537
C08478=1198.164,415.528,-84.146,-175.881,8.680,148.537
C08479=1198.168,415.282,-84.111,-175.881,8.678,148.536
C08480=1198.172,415.034,-84.075,-175.882,8.676,148.535
C08481=1198.175,414.787,-84.039,-175.882,8.673,148.535
C08482=1198.179,414.540,-84.004,-175.882,8.671,148.534
C08483=1198.183,414.292,-83.969,-175.882,8.669,148.534
C08484=1198.188,414.045,-83.933,-175.882,8.668,148.534
C08485=1198.192,413.796,-83.898,-175.883,8.666,148.533
C08486=1198.196,413.550,-83.863,-175.883,8.663,148.533
C08487=1198.199,413.302,-83.827,-175.883,8.661,148.532
C08488=1198.203,413.055,-83.791,-175.883,8.659,148.532
C08489=1198.207,412.808,-83.756,-175.884,8.656,148.531
C08490=1198.211,412.560,-83.721,-175.884,8.654,148.530
C08491=1198.215,412.312,-83.686,-175.883,8.653,148.530
C08492=1198.219,412.064,-83.650,-175.884,8.651,148.530
C08493=1198.224,411.818,-83.615,-175.884,8.649,148.529
C08494=1198.227,411.570,-83.579,-175.885,8.646,148.529
C08495=1198.231,411.323,-83.543,-175.885,8.644,148.528
C08496=1198.236,411.075,-83.509,-175.885,8.642,148.528
C08497=1198.239,410.828,-83.473,-175.885,8.639,148.527
C08498=1198.243,410.580,-83.438,-175.886,8.637,148.526
C08499=1198.247,410.333,-83.402,-175.886,8.635,148.526
C08500=1198.251,410.086,-83.367,-175.886,8.633,148.525
C08501=1198.256,409.837,-83.332,-175.886,8.630,148.525
C08502=1198.259,409.590,-83.296,-175.887,8.628,148.525
C08503=1198.263,409.343,-83.261,-175.887,8.626,148.524
C08504=1198.267,409.096,-83.225,-175.887,8.625,148.524
C08505=1198.271,408.848,-83.191,-175.887,8.622,148.523
C08506=1198.275,408.601,-83.155,-175.887,8.620,148.523
C08507=1198.279,408.353,-83.120,-175.888,8.618,148.522
C08508=1198.283,408.106,-83.084,-175.888,8.616,148.521
C08509=1198.287,407.858,-83.050,-175.888,8.613,148.521
C08510=1198.291,407.611,-83.014,-175.888,8.611,148.520
C08511=1198.295,407.363,-82.979,-175.889,8.609,148.520
C08512=1198.298,407.116,-82.943,-175.889,8.607,148.519
C08513=1198.303,406.868,-82.909,-175.889,8.604,148.519
C08514=1198.307,406.621,-82.873,-175.889,8.602,148.518
C08515=1198.311,406.373,-82.837,-175.889,8.600,148.518
C08516=1198.315,406.126,-82.803,-175.890,8.597,148.517
C08517=1198.319,405.878,-82.767,-175.890,8.594,148.517
C08518=1198.323,405.631,-82.732,-175.891,8.592,148.516
C08519=1198.327,405.383,-82.697,-175.891,8.590,148.516
C08520=1198.331,405.136,-82.662,-175.892,8.588,148.515
C08521=1198.335,404.888,-82.626,-175.892,8.586,148.515
C08522=1198.339,404.641,-82.592,-175.892,8.583,148.514
C08523=1198.343,404.393,-82.556,-175.892,8.581,148.514
C08524=1198.347,404.146,-82.520,-175.893,8.579,148.513
C08525=1198.351,403.898,-82.486,-175.893,8.577,148.513
C08526=1198.355,403.651,-82.450,-175.893,8.574,148.512
C08527=1198.359,403.404,-82.415,-175.893,8.572,148.512
C08528=1198.363,403.156,-82.380,-175.894,8.569,148.511
C08529=1198.367,402.908,-82.345,-175.894,8.567,148.510
C08530=1198.371,402.662,-82.310,-175.894,8.564,148.510
C08531=1198.375,402.414,-82.275,-175.895,8.562,148.509
C08532=1198.379,402.166,-82.239,-175.895,8.560,148.509
C08533=1198.383,401.919,-82.205,-175.895,8.558,148.508
C08534=1198.387,401.671,-82.169,-175.895,8.555,148.508
C08535=1198.390,401.424,-82.134,-175.896,8.552,148.507
C08536=1198.395,401.176,-82.099,-175.896,8.550,148.507
C08537=1198.399,400.929,-82.064,-175.897,8.548,148.506
C08538=1198.403,400.681,-82.029,-175.897,8.545,148.506
C08539=1198.407,400.434,-81.994,-175.897,8.543,148.505
C08540=1198.411,400.186,-81.958,-175.898,8.540,148.504
C08541=1198.415,399.939,-81.924,-175.898,8.538,148.504
C08542=1198.419,399.691,-81.888,-175.898,8.536,148.503
C08543=1198.423,399.443,-81.853,-175.899,8.533,148.503
C08544=1198.427,399.196,-81.818,-175.899,8.530,148.502
C08545=1198.431,398.948,-81.783,-175.900,8.528,148.502
C08546=1198.435,398.702,-81.748,-175.900,8.526,148.501
C08547=1198.439,398.453,-81.713,-175.900,8.523,148.501
C08548=1198.443,398.206,-81.678,-175.901,8.520,148.500
C08549=1198.447,397.958,-81.643,-175.901,8.518,148.500
C08550=1198.451,397.711,-81.608,-175.901,8.516,148.499
C08551=1198.455,397.464,-81.574,-175.903,8.513,148.499
C08552=1198.459,397.216,-81.538,-175.903,8.511,148.498
C08553=1198.463,396.968,-81.503,-175.903,8.508,148.498
C08554=1198.467,396.721,-81.468,-175.904,8.505,148.497
C08555=1198.471,396.473,-81.433,-175.904,8.503,148.496
C08556=1198.475,396.227,-81.398,-175.904,8.501,148.496
C08557=1198.479,395.978,-81.363,-175.905,8.498,148.495
C08558=1198.483,395.731,-81.328,-175.905,8.495,148.495
C08559=1198.487,395.484,-81.293,-175.906,8.492,148.494
C08560=1198.491,395.236,-81.258,-175.906,8.490,148.494
C08561=1198.496,394.989,-81.223,-175.907,8.488,148.493
C08562=1198.499,394.741,-81.188,-175.907,8.485,148.493
C08563=1198.503,394.494,-81.154,-175.908,8.482,148.492
C08564=1198.507,394.246,-81.119,-175.908,8.479,148.491
C08565=1198.511,393.998,-81.084,-175.909,8.477,148.491
C08566=1198.515,393.751,-81.049,-175.909,8.474,148.490
C08567=1198.519,393.503,-81.014,-175.910,8.472,148.490
C08568=1198.523,393.256,-80.979,-175.910,8.469,148.489
C08569=1198.527,393.008,-80.944,-175.911,8.466,148.489
C08570=1198.532,392.726,-80.904,-175.911,8.463,148.488
C08571=1198.536,392.443,-80.865,-175.912,8.460,148.488
C08572=1198.541,392.159,-80.825,-175.913,8.457,148.487
C08573=1198.545,391.877,-80.785,-175.914,8.454,148.486
C08574=1198.550,391.629,-80.750,-175.914,8.452,148.486
C08575=1198.554,391.381,-80.715,-175.915,8.449,148.485
C08576=1198.557,391.134,-80.680,-175.915,8.446,148.485
C08577=1198.562,390.886,-80.645,-175.916,8.443,148.484
C08578=1198.565,390.639,-80.611,-175.916,8.440,148.484
C08579=1198.569,390.392,-80.576,-175.917,8.438,148.483
C08580=1198.573,390.144,-80.541,-175.918,8.435,148.483
C08581=1198.578,389.896,-80.507,-175.918,8.433,148.482
C08582=1198.581,389.649,-80.471,-175.919,8.430,148.481
C08583=1198.585,389.402,-80.437,-175.920,8.427,148.481
C08584=1198.589,389.153,-80.402,-175.920,8.424,148.480
C08585=1198.594,388.906,-80.368,-175.921,8.421,148.480
C08586=1198.598,388.659,-80.332,-175.922,8.418,148.479
C08587=1198.602,388.411,-80.298,-175.922,8.416,148.479
C08588=1198.605,388.163,-80.264,-175.923,8.413,148.478
C08589=1198.610,387.917,-80.229,-175.924,8.410,148.478
C08590=1198.614,387.668,-80.194,-175.925,8.407,148.477
C08591=1198.618,387.421,-80.159,-175.925,8.404,148.477
C08592=1198.621,387.173,-80.125,-175.926,8.402,148.476
C08593=1198.626,386.926,-80.091,-175.927,8.399,148.476
C08594=1198.630,386.678,-80.055,-175.928,8.395,148.475
C08595=1198.634,386.431,-80.021,-175.928,8.393,148.474
C08596=1198.637,386.183,-79.986,-175.929,8.390,148.474
C08597=1198.642,385.936,-79.952,-175.930,8.387,148.473
C08598=1198.646,385.688,-79.917,-175.931,8.384,148.473
C08599=1198.650,385.441,-79.882,-175.931,8.381,148.472
C08600=1198.653,385.193,-79.848,-175.932,8.379,148.472
C08601=1198.658,384.945,-79.813,-175.933,8.376,148.471
C08602=1198.662,384.697,-79.778,-175.934,8.373,148.471
C08603=1198.667,384.450,-79.744,-175.934,8.370,148.470
C08604=1198.670,384.202,-79.710,-175.936,8.367,148.470
C08605=1198.674,383.955,-79.675,-175.936,8.364,148.469
C08606=1198.678,383.707,-79.640,-175.937,8.361,148.469
C08607=1198.682,383.460,-79.606,-175.938,8.358,148.468
C08608=1198.686,383.213,-79.571,-175.939,8.355,148.468
C08609=1198.690,382.965,-79.536,-175.940,8.352,148.467
C08610=1198.694,382.717,-79.503,-175.941,8.350,148.467
C08611=1198.698,382.469,-79.468,-175.941,8.347,148.466
C08612=1198.703,382.222,-79.433,-175.943,8.344,148.466
C08613=1198.706,381.974,-79.399,-175.943,8.341,148.465
C08614=1198.711,381.727,-79.365,-175.944,8.338,148.465
C08615=1198.714,381.479,-79.330,-175.945,8.335,148.464
C08616=1198.718,381.231,-79.296,-175.946,8.332,148.464
C08617=1198.723,380.984,-79.261,-175.947,8.329,148.463
C08618=1198.727,380.736,-79.227,-175.948,8.326,148.463
C08619=1198.731,380.489,-79.193,-175.950,8.322,148.462
C08620=1198.735,380.241,-79.158,-175.951,8.319,148.462
C08621=1198.738,379.994,-79.124,-175.952,8.316,148.461
C08622=1198.743,379.746,-79.089,-175.953,8.313,148.461
C08623=1198.747,379.498,-79.055,-175.954,8.310,148.460
C08624=1198.751,379.251,-79.021,-175.955,8.307,148.460
C08625=1198.755,379.003,-78.986,-175.956,8.305,148.459
C08626=1198.759,378.756,-78.952,-175.957,8.301,148.459
C08627=1198.763,378.508,-78.918,-175.958,8.299,148.458
C08628=1198.767,378.260,-78.883,-175.959,8.296,148.458
C08629=1198.771,378.013,-78.849,-175.960,8.293,148.457
C08630=1198.775,377.765,-78.814,-175.962,8.289,148.457
C08631=1198.779,377.518,-78.780,-175.962,8.286,148.456
C08632=1198.783,377.270,-78.746,-175.964,8.283,148.456
C08633=1198.787,377.023,-78.712,-175.964,8.280,148.455
C08634=1198.792,376.775,-78.678,-175.966,8.277,148.455
C08635=1198.795,376.527,-78.644,-175.967,8.274,148.454
C08636=1198.799,376.279,-78.609,-175.968,8.271,148.454
C08637=1198.804,376.032,-78.575,-175.970,8.268,148.453
C08638=1198.807,375.784,-78.540,-175.971,8.265,148.453
C08639=1198.812,375.537,-78.506,-175.971,8.262,148.452
C08640=1198.816,375.290,-78.472,-175.973,8.258,148.452
C08641=1198.820,375.041,-78.438,-175.975,8.255,148.452
C08642=1198.824,374.794,-78.404,-175.975,8.252,148.451
C08643=1198.827,374.547,-78.370,-175.976,8.249,148.451
C08644=1198.831,374.298,-78.335,-175.978,8.246,148.450
C08645=1198.835,374.051,-78.301,-175.980,8.243,148.450
C08646=1198.840,373.803,-78.268,-175.981,8.240,148.449
C08647=1198.843,373.556,-78.233,-175.981,8.237,148.449
C08648=1198.848,373.308,-78.199,-175.983,8.233,148.448
C08649=1198.852,373.061,-78.165,-175.985,8.231,148.448
C08650=1198.856,372.812,-78.131,-175.986,8.228,148.448
C08651=1198.860,372.565,-78.097,-175.988,8.224,148.447
C08652=1198.864,372.318,-78.063,-175.988,8.221,148.447
C08653=1198.868,372.069,-78.029,-175.989,8.218,148.446
C08654=1198.872,371.822,-77.995,-175.991,8.215,148.446
C08655=1198.876,371.575,-77.961,-175.992,8.212,148.445
C08656=1198.881,371.327,-77.928,-175.994,8.209,148.445
C08657=1198.884,371.079,-77.893,-175.996,8.205,148.445
C08658=1198.888,370.832,-77.859,-175.997,8.203,148.444
C08659=1198.892,370.584,-77.826,-175.999,8.199,148.444
C08660=1198.896,370.336,-77.791,-176.000,8.196,148.443
C08661=1198.900,370.089,-77.757,-176.001,8.193,148.443
C08662=1198.905,369.841,-77.723,-176.003,8.190,148.443
C08663=1198.909,369.594,-77.689,-176.004,8.187,148.442
C08664=1198.912,369.345,-77.656,-176.006,8.183,148.442
C08665=1198.917,369.098,-77.621,-176.007,8.181,148.441
C08666=1198.921,368.851,-77.588,-176.009,8.177,148.441
C08667=1198.925,368.603,-77.554,-176.010,8.174,148.440
C08668=1198.929,368.355,-77.520,-176.011,8.171,148.440
C08669=1198.933,368.107,-77.486,-176.013,8.168,148.440
C08670=1198.937,367.860,-77.453,-176.014,8.165,148.439
C08671=1198.942,367.612,-77.419,-176.016,8.161,148.439
C08672=1198.945,367.364,-77.385,-176.017,8.158,148.438
C08673=1198.949,367.116,-77.351,-176.019,8.155,148.438
C08674=1198.954,366.836,-77.313,-176.021,8.151,148.438
C08675=1198.959,366.555,-77.274,-176.022,8.147,148.437
C08676=1198.964,366.274,-77.237,-176.024,8.144,148.437
C08677=1198.968,365.994,-77.199,-176.026,8.140,148.436
C08678=1198.972,365.746,-77.164,-176.027,8.137,148.436
C08679=1198.976,365.498,-77.131,-176.029,8.134,148.436
C08680=1198.980,365.251,-77.097,-176.031,8.131,148.435
C08681=1198.984,365.003,-77.064,-176.032,8.128,148.435
C08682=1198.989,364.755,-77.030,-176.034,8.125,148.434
C08683=1198.993,364.508,-76.996,-176.036,8.121,148.434
C08684=1198.996,364.259,-76.963,-176.037,8.119,148.434
C08685=1199.000,364.012,-76.929,-176.039,8.115,148.433
C08686=1199.004,363.765,-76.896,-176.041,8.111,148.433
C08687=1199.009,363.517,-76.862,-176.042,8.109,148.433
C08688=1199.013,363.269,-76.829,-176.044,8.105,148.432
C08689=1199.017,363.022,-76.795,-176.045,8.102,148.432
C08690=1199.020,362.773,-76.761,-176.048,8.099,148.432
C08691=1199.025,362.526,-76.728,-176.049,8.096,148.431
C08692=1199.028,362.278,-76.694,-176.051,8.093,148.431
C08693=1199.033,362.030,-76.661,-176.053,8.089,148.431
C08694=1199.037,361.783,-76.627,-176.054,8.087,148.430
C08695=1199.042,361.535,-76.594,-176.056,8.083,148.430
C08696=1199.045,361.287,-76.560,-176.058,8.080,148.430
C08697=1199.049,361.039,-76.527,-176.059,8.077,148.429
C08698=1199.053,360.792,-76.494,-176.062,8.073,148.429
C08699=1199.057,360.544,-76.461,-176.063,8.071,148.429
C08700=1199.061,360.296,-76.427,-176.064,8.067,148.428
C08701=1199.066,360.049,-76.393,-176.067,8.064,148.428
C08702=1199.070,359.801,-76.360,-176.068,8.061,148.428
C08703=1199.074,359.553,-76.327,-176.070,8.058,148.427
C08704=1199.078,359.306,-76.293,-176.072,8.054,148.427
C08705=1199.082,359.057,-76.260,-176.074,8.051,148.427
C08706=1199.086,358.809,-76.227,-176.075,8.048,148.426
C08707=1199.090,358.562,-76.193,-176.078,8.044,148.426
C08708=1199.094,358.315,-76.160,-176.079,8.042,148.426
C08709=1199.098,358.067,-76.127,-176.081,8.038,148.425
C08710=1199.102,357.819,-76.093,-176.083,8.035,148.425
C08711=1199.106,357.571,-76.060,-176.085,8.032,148.425
C08712=1199.111,357.324,-76.027,-176.087,8.029,148.425
C08713=1199.115,357.076,-75.994,-176.089,8.025,148.424
C08714=1199.119,356.828,-75.961,-176.090,8.023,148.424
C08715=1199.123,356.581,-75.928,-176.092,8.019,148.424
C08716=1199.127,356.333,-75.894,-176.094,8.016,148.423
C08717=1199.131,356.085,-75.861,-176.096,8.013,148.423
C08718=1199.135,355.837,-75.828,-176.098,8.010,148.423
C08719=1199.139,355.589,-75.795,-176.100,8.006,148.422
C08720=1199.143,355.341,-75.761,-176.102,8.004,148.422
C08721=1199.147,355.093,-75.728,-176.103,8.000,148.422
C08722=1199.151,354.846,-75.695,-176.106,7.997,148.422
C08723=1199.155,354.598,-75.662,-176.107,7.994,148.421
C08724=1199.160,354.350,-75.629,-176.109,7.991,148.421
C08725=1199.164,354.103,-75.596,-176.111,7.987,148.421
C08726=1199.168,353.854,-75.563,-176.113,7.984,148.421
C08727=1199.172,353.606,-75.530,-176.115,7.981,148.420
C08728=1199.176,353.359,-75.497,-176.117,7.978,148.420
C08729=1199.180,353.111,-75.464,-176.119,7.974,148.420
C08730=1199.184,352.864,-75.431,-176.121,7.972,148.420
C08731=1199.188,352.616,-75.398,-176.123,7.969,148.419
C08732=1199.192,352.368,-75.365,-176.125,7.965,148.419
C08733=1199.197,352.120,-75.332,-176.126,7.962,148.419
C08734=1199.201,351.872,-75.299,-176.129,7.959,148.418
C08735=1199.206,351.625,-75.267,-176.131,7.956,148.418
C08736=1199.210,351.377,-75.233,-176.133,7.952,148.418
C08737=1199.213,351.129,-75.202,-176.134,7.950,148.418
C08738=1199.218,350.882,-75.168,-176.137,7.946,148.417
C08739=1199.222,350.634,-75.135,-176.139,7.943,148.417
C08740=1199.226,350.386,-75.102,-176.140,7.940,148.417
C08741=1199.230,350.138,-75.070,-176.143,7.937,148.417
C08742=1199.234,349.890,-75.036,-176.145,7.934,148.417
C08743=1199.238,349.643,-75.004,-176.147,7.931,148.416
C08744=1199.242,349.394,-74.971,-176.148,7.928,148.416
C08745=1199.246,349.146,-74.938,-176.151,7.924,148.416
C08746=1199.251,348.899,-74.905,-176.153,7.921,148.415
C08747=1199.254,348.651,-74.873,-176.154,7.918,148.415
C08748=1199.258,348.403,-74.840,-176.157,7.915,148.415
C08749=1199.263,348.156,-74.807,-176.159,7.912,148.415
C08750=1199.268,347.908,-74.775,-176.161,7.909,148.415
C08751=1199.271,347.660,-74.742,-176.163,7.906,148.414
C08752=1199.275,347.412,-74.710,-176.165,7.903,148.414
C08753=1199.280,347.164,-74.677,-176.167,7.899,148.414
C08754=1199.284,346.916,-74.644,-176.169,7.897,148.414
C08755=1199.287,346.668,-74.612,-176.171,7.893,148.414
C08756=1199.292,346.421,-74.579,-176.173,7.890,148.413
C08757=1199.297,346.173,-74.547,-176.175,7.888,148.413
C08758=1199.300,345.926,-74.514,-176.177,7.884,148.413
C08759=1199.304,345.677,-74.482,-176.180,7.881,148.413
C08760=1199.309,345.429,-74.448,-176.182,7.878,148.413
C08761=1199.312,345.181,-74.417,-176.183,7.875,148.412
C08762=1199.316,344.934,-74.383,-176.186,7.872,148.412
C08763=1199.321,344.685,-74.351,-176.188,7.868,148.412
C08764=1199.325,344.438,-74.319,-176.190,7.866,148.412
C08765=1199.329,344.190,-74.286,-176.192,7.863,148.412
C08766=1199.334,343.942,-74.254,-176.194,7.859,148.411
C08767=1199.337,343.695,-74.221,-176.196,7.856,148.411
C08768=1199.342,343.446,-74.189,-176.198,7.853,148.411
C08769=1199.347,343.199,-74.157,-176.200,7.850,148.411
C08770=1199.350,342.951,-74.124,-176.202,7.847,148.410
C08771=1199.354,342.703,-74.092,-176.204,7.844,148.410
C08772=1199.358,342.455,-74.059,-176.206,7.841,148.410
C08773=1199.362,342.207,-74.027,-176.209,7.838,148.410
C08774=1199.367,341.959,-73.995,-176.211,7.835,148.410
C08775=1199.371,341.711,-73.963,-176.213,7.832,148.410
C08776=1199.375,341.464,-73.930,-176.215,7.829,148.409
C08777=1199.379,341.216,-73.898,-176.217,7.825,148.409
C08778=1199.384,340.938,-73.862,-176.220,7.822,148.409
C08779=1199.388,340.659,-73.825,-176.222,7.819,148.409
C08780=1199.393,340.380,-73.789,-176.224,7.816,148.409
C08781=1199.398,340.102,-73.753,-176.227,7.812,148.409
C08782=1199.402,339.854,-73.721,-176.229,7.809,148.408
C08783=1199.406,339.606,-73.688,-176.231,7.806,148.408
C08784=1199.410,339.358,-73.656,-176.233,7.802,148.408
C08785=1199.415,339.111,-73.624,-176.235,7.800,148.408
C08786=1199.419,338.863,-73.592,-176.238,7.797,148.408
C08787=1199.423,338.614,-73.560,-176.240,7.793,148.407
C08788=1199.427,338.367,-73.528,-176.242,7.790,148.407
C08789=1199.431,338.119,-73.495,-176.244,7.788,148.407
C08790=1199.435,337.871,-73.463,-176.246,7.785,148.407
C08791=1199.439,337.623,-73.432,-176.249,7.781,148.407
C08792=1199.444,337.375,-73.399,-176.250,7.779,148.407
C08793=1199.448,337.127,-73.368,-176.253,7.775,148.406
C08794=1199.452,336.879,-73.335,-176.255,7.772,148.406
C08795=1199.456,336.632,-73.304,-176.258,7.769,148.406
C08796=1199.460,336.384,-73.272,-176.259,7.767,148.406
C08797=1199.464,336.135,-73.239,-176.261,7.763,148.406
C08798=1199.469,335.888,-73.208,-176.264,7.760,148.406
C08799=1199.473,335.640,-73.175,-176.266,7.758,148.406
C08800=1199.477,335.392,-73.144,-176.268,7.754,148.405
C08801=1199.481,335.144,-73.112,-176.271,7.751,148.405
C08802=1199.486,334.896,-73.080,-176.273,7.748,148.405
C08803=1199.489,334.648,-73.048,-176.275,7.745,148.405
C08804=1199.494,334.401,-73.016,-176.277,7.742,148.405
C08805=1199.498,334.152,-72.984,-176.279,7.739,148.405
C08806=1199.502,333.904,-72.952,-176.282,7.736,148.405
C08807=1199.506,333.657,-72.921,-176.284,7.734,148.405
C08808=1199.510,333.409,-72.889,-176.286,7.730,148.404
C08809=1199.514,333.160,-72.856,-176.288,7.727,148.404
C08810=1199.519,332.912,-72.826,-176.290,7.725,148.404
C08811=1199.523,332.664,-72.794,-176.293,7.721,148.404
C08812=1199.528,332.417,-72.762,-176.295,7.718,148.404
C08813=1199.531,332.169,-72.730,-176.298,7.715,148.404
C08814=1199.535,331.921,-72.698,-176.299,7.713,148.404
C08815=1199.539,331.673,-72.666,-176.302,7.709,148.404
C08816=1199.544,331.424,-72.635,-176.304,7.706,148.403
C08817=1199.548,331.177,-72.603,-176.306,7.704,148.403
C08818=1199.552,330.929,-72.571,-176.309,7.701,148.403
C08819=1199.556,330.681,-72.540,-176.311,7.697,148.403
C08820=1199.560,330.434,-72.508,-176.313,7.694,148.403
C08821=1199.565,330.185,-72.476,-176.315,7.692,148.403
C08822=1199.569,329.937,-72.445,-176.317,7.688,148.403
C08823=1199.573,329.689,-72.413,-176.320,7.685,148.403
C08824=1199.578,329.441,-72.382,-176.322,7.682,148.402
C08825=1199.581,329.193,-72.350,-176.324,7.680,148.403
C08826=1199.585,328.945,-72.319,-176.327,7.677,148.402
C08827=1199.590,328.697,-72.287,-176.329,7.674,148.402
C08828=1199.594,328.449,-72.255,-176.331,7.671,148.402
C08829=1199.598,328.202,-72.224,-176.334,7.668,148.402
C08830=1199.602,327.953,-72.193,-176.336,7.665,148.402
C08831=1199.607,327.706,-72.161,-176.339,7.662,148.402
C08832=1199.610,327.458,-72.129,-176.340,7.659,148.402
C08833=1199.615,327.210,-72.099,-176.343,7.656,148.402
C08834=1199.619,326.962,-72.067,-176.345,7.653,148.402
C08835=1199.624,326.713,-72.035,-176.347,7.651,148.402
C08836=1199.628,326.465,-72.004,-176.349,7.647,148.401
C08837=1199.632,326.217,-71.973,-176.352,7.644,148.401
C08838=1199.636,325.969,-71.941,-176.354,7.641,148.401
C08839=1199.641,325.721,-71.910,-176.357,7.639,148.401
C08840=1199.644,325.473,-71.878,-176.359,7.635,148.401
C08841=1199.649,325.225,-71.848,-176.361,7.632,148.401
C08842=1199.653,324.977,-71.816,-176.363,7.630,148.401
C08843=1199.657,324.729,-71.785,-176.366,7.627,148.401
C08844=1199.661,324.481,-71.753,-176.368,7.624,148.401
C08845=1199.666,324.233,-71.722,-176.371,7.620,148.401
C08846=1199.669,323.985,-71.691,-176.373,7.618,148.401
C08847=1199.674,323.737,-71.660,-176.375,7.615,148.400
C08848=1199.678,323.490,-71.628,-176.378,7.612,148.400
C08849=1199.682,323.241,-71.597,-176.379,7.609,148.400
C08850=1199.687,322.993,-71.566,-176.382,7.606,148.400
C08851=1199.691,322.745,-71.535,-176.385,7.603,148.400
C08852=1199.695,322.497,-71.504,-176.387,7.600,148.400
C08853=1199.699,322.249,-71.473,-176.389,7.598,148.400
C08854=1199.703,322.002,-71.442,-176.391,7.594,148.400
C08855=1199.707,321.754,-71.411,-176.394,7.591,148.400
C08856=1199.711,321.505,-71.380,-176.396,7.589,148.400
C08857=1199.716,321.258,-71.348,-176.398,7.586,148.400
C08858=1199.720,321.009,-71.317,-176.401,7.583,148.400
C08859=1199.724,320.761,-71.287,-176.403,7.580,148.400
C08860=1199.729,320.514,-71.255,-176.405,7.577,148.400
C08861=1199.733,320.265,-71.224,-176.408,7.574,148.400
C08862=1199.737,320.017,-71.193,-176.410,7.571,148.399
C08863=1199.741,319.769,-71.163,-176.413,7.569,148.399
C08864=1199.745,319.521,-71.132,-176.415,7.566,148.399
C08865=1199.749,319.274,-71.100,-176.417,7.562,148.399
C08866=1199.753,319.025,-71.069,-176.420,7.559,148.399
C08867=1199.758,318.777,-71.039,-176.422,7.557,148.399
C08868=1199.763,318.529,-71.008,-176.425,7.554,148.399
C08869=1199.766,318.281,-70.977,-176.427,7.551,148.399
C08870=1199.771,318.033,-70.946,-176.429,7.549,148.399
C08871=1199.775,317.785,-70.915,-176.432,7.545,148.399
C08872=1199.779,317.537,-70.884,-176.434,7.542,148.399
C08873=1199.784,317.289,-70.853,-176.436,7.540,148.399
C08874=1199.787,317.041,-70.823,-176.439,7.537,148.399
C08875=1199.791,316.792,-70.792,-176.441,7.534,148.399
C08876=1199.796,316.544,-70.761,-176.444,7.531,148.399
C08877=1199.801,316.296,-70.730,-176.446,7.529,148.399
C08878=1199.804,316.048,-70.700,-176.448,7.525,148.399
C08879=1199.809,315.800,-70.669,-176.451,7.522,148.399
C08880=1199.813,315.552,-70.638,-176.453,7.520,148.399
C08881=1199.817,315.304,-70.607,-176.456,7.517,148.399
C08882=1199.822,315.028,-70.573,-176.458,7.514,148.399
C08883=1199.827,314.751,-70.539,-176.461,7.511,148.399
C08884=1199.831,314.475,-70.505,-176.463,7.508,148.399
C08885=1199.836,314.199,-70.470,-176.466,7.505,148.399
C08886=1199.840,313.951,-70.441,-176.469,7.502,148.399
C08887=1199.845,313.703,-70.410,-176.472,7.499,148.399
C08888=1199.849,313.454,-70.379,-176.474,7.495,148.398
C08889=1199.853,313.207,-70.349,-176.476,7.493,148.398
C08890=1199.857,312.959,-70.318,-176.479,7.490,148.398
C08891=1199.862,312.711,-70.287,-176.481,7.487,148.398
C08892=1199.865,312.462,-70.257,-176.483,7.484,148.398
C08893=1199.870,312.214,-70.226,-176.486,7.481,148.398
C08894=1199.874,311.966,-70.197,-176.488,7.478,148.398
C08895=1199.879,311.718,-70.166,-176.490,7.476,148.398
C08896=1199.883,311.470,-70.135,-176.493,7.473,148.398
C08897=1199.886,311.222,-70.104,-176.495,7.470,148.398
C08898=1199.891,310.974,-70.074,-176.498,7.468,148.398
C08899=1199.895,310.726,-70.044,-176.500,7.465,148.398
C08900=1199.900,310.478,-70.013,-176.503,7.462,148.398
C08901=1199.904,310.230,-69.983,-176.505,7.459,148.398
C08902=1199.908,309.981,-69.952,-176.508,7.456,148.398
C08903=1199.913,309.733,-69.922,-176.510,7.453,148.398
C08904=1199.917,309.485,-69.892,-176.512,7.451,148.398
C08905=1199.921,309.237,-69.861,-176.515,7.448,148.398
C08906=1199.925,308.989,-69.832,-176.517,7.445,148.398
C08907=1199.930,308.741,-69.801,-176.520,7.442,148.398
C08908=1199.933,308.493,-69.770,-176.522,7.440,148.398
C08909=1199.938,308.244,-69.740,-176.525,7.436,148.398
C08910=1199.942,307.996,-69.710,-176.527,7.433,148.398
C08911=1199.947,307.748,-69.679,-176.529,7.431,148.398
C08912=1199.951,307.500,-69.650,-176.532,7.428,148.398
C08913=1199.955,307.252,-69.619,-176.535,7.425,148.398
C08914=1199.960,307.004,-69.590,-176.537,7.423,148.398
C08915=1199.963,306.756,-69.560,-176.540,7.420,148.398
C08916=1199.968,306.507,-69.529,-176.542,7.417,148.398
C08917=1199.972,306.259,-69.499,-176.544,7.414,148.398
C08918=1199.976,306.011,-69.468,-176.547,7.411,148.398
C08919=1199.980,305.763,-69.439,-176.549,7.408,148.398
C08920=1199.985,305.515,-69.408,-176.551,7.406,148.398
C08921=1199.989,305.267,-69.379,-176.554,7.403,148.398
C08922=1199.993,305.019,-69.348,-176.557,7.400,148.398
C08923=1199.998,304.771,-69.318,-176.559,7.398,148.398
C08924=1200.002,304.522,-69.289,-176.562,7.395,148.398
C08925=1200.007,304.274,-69.258,-176.564,7.393,148.398
C08926=1200.011,304.026,-69.229,-176.567,7.390,148.398
C08927=1200.015,303.778,-69.199,-176.569,7.386,148.398
C08928=1200.020,303.530,-69.168,-176.571,7.384,148.398
C08929=1200.023,303.282,-69.138,-176.574,7.381,148.398
C08930=1200.027,303.033,-69.108,-176.576,7.378,148.398
C08931=1200.032,302.785,-69.078,-176.578,7.376,148.398
C08932=1200.036,302.537,-69.048,-176.581,7.373,148.398
C08933=1200.040,302.289,-69.019,-176.584,7.370,148.398
C08934=1200.045,302.040,-68.989,-176.586,7.368,148.398
C08935=1200.049,301.793,-68.959,-176.589,7.365,148.398
C08936=1200.053,301.544,-68.929,-176.591,7.362,148.398
C08937=1200.057,301.296,-68.900,-176.593,7.359,148.398
C08938=1200.062,301.047,-68.870,-176.596,7.356,148.398
C08939=1200.066,300.800,-68.839,-176.599,7.353,148.398
C08940=1200.070,300.552,-68.810,-176.601,7.351,148.399
C08941=1200.075,300.303,-68.781,-176.604,7.348,148.399
C08942=1200.080,300.055,-68.751,-176.606,7.346,148.399
C08943=1200.083,299.807,-68.720,-176.608,7.343,148.399
C08944=1200.088,299.559,-68.691,-176.611,7.340,148.399
C08945=1200.092,299.310,-68.661,-176.613,7.338,148.399
C08946=1200.096,299.062,-68.632,-176.616,7.335,148.399
C08947=1200.101,298.814,-68.602,-176.619,7.332,148.399
C08948=1200.105,298.566,-68.572,-176.621,7.330,148.399
C08949=1200.109,298.318,-68.542,-176.624,7.327,148.399
C08950=1200.114,298.070,-68.513,-176.626,7.324,148.399
C08951=1200.118,297.822,-68.484,-176.628,7.321,148.399
C08952=1200.122,297.574,-68.454,-176.631,7.318,148.399
C08953=1200.127,297.325,-68.424,-176.633,7.316,148.399
C08954=1200.131,297.077,-68.395,-176.636,7.313,148.399
C08955=1200.135,296.829,-68.365,-176.639,7.310,148.399
C08956=1200.140,296.580,-68.336,-176.641,7.308,148.399
C08957=1200.144,296.332,-68.306,-176.643,7.305,148.399
C08958=1200.148,296.084,-68.277,-176.646,7.303,148.399
C08959=1200.152,295.835,-68.248,-176.648,7.300,148.399
C08960=1200.156,295.587,-68.218,-176.651,7.297,148.399
C08961=1200.160,295.339,-68.189,-176.653,7.294,148.399
C08962=1200.165,295.091,-68.159,-176.656,7.291,148.399
C08963=1200.169,294.843,-68.130,-176.659,7.288,148.399
C08964=1200.174,294.595,-68.101,-176.661,7.286,148.399
C08965=1200.178,294.346,-68.071,-176.663,7.283,148.399
C08966=1200.183,294.098,-68.041,-176.665,7.281,148.399
C08967=1200.187,293.850,-68.012,-176.668,7.278,148.400
C08968=1200.191,293.601,-67.982,-176.671,7.275,148.400
C08969=1200.195,293.353,-67.953,-176.673,7.273,148.400
C08970=1200.199,293.105,-67.923,-176.676,7.270,148.400
C08971=1200.204,292.857,-67.894,-176.678,7.268,148.400
C08972=1200.208,292.609,-67.865,-176.681,7.265,148.400
C08973=1200.213,292.360,-67.836,-176.684,7.262,148.400
C08974=1200.217,292.112,-67.807,-176.686,7.260,148.400
C08975=1200.220,291.864,-67.778,-176.689,7.257,148.400
C08976=1200.225,291.616,-67.748,-176.691,7.255,148.400
C08977=1200.229,291.368,-67.719,-176.693,7.252,148.400
C08978=1200.234,291.120,-67.690,-176.696,7.248,148.400
C08979=1200.238,290.871,-67.661,-176.698,7.246,148.400
C08980=1200.242,290.623,-67.632,-176.701,7.243,148.400
C08981=1200.246,290.374,-67.602,-176.703,7.241,148.400
C08982=1200.251,290.126,-67.573,-176.706,7.238,148.400
C08983=1200.256,289.878,-67.544,-176.708,7.236,148.401
C08984=1200.260,289.630,-67.515,-176.711,7.233,148.401
C08985=1200.264,289.381,-67.485,-176.714,7.230,148.401
C08986=1200.269,289.107,-67.454,-176.716,7.227,148.401
C08987=1200.274,288.833,-67.422,-176.719,7.224,148.401
C08988=1200.278,288.559,-67.390,-176.722,7.221,148.401
C08989=1200.283,288.284,-67.357,-176.724,7.219,148.401
C08990=1200.288,288.036,-67.328,-176.727,7.216,148.401
C08991=1200.292,287.787,-67.300,-176.730,7.213,148.401
C08992=1200.296,287.539,-67.270,-176.732,7.211,148.401
C08993=1200.300,287.290,-67.242,-176.735,7.208,148.401
C08994=1200.305,287.043,-67.213,-176.737,7.206,148.401
C08995=1200.309,286.794,-67.183,-176.740,7.203,148.401
C08996=1200.313,286.546,-67.155,-176.742,7.201,148.402
C08997=1200.317,286.298,-67.126,-176.745,7.198,148.402
C08998=1200.322,286.049,-67.097,-176.748,7.195,148.402
C08999=1200.327,285.801,-67.068,-176.750,7.193,148.402
C09000=1200.330,285.553,-67.040,-176.752,7.190,148.402
C09001=1200.335,285.305,-67.011,-176.755,7.188,148.402
C09002=1200.340,285.056,-66.982,-176.758,7.185,148.402
C09003=1200.344,284.808,-66.952,-176.760,7.183,148.402
C09004=1200.348,284.560,-66.925,-176.763,7.180,148.402
C09005=1200.352,284.312,-66.895,-176.765,7.177,148.402
C09006=1200.357,284.063,-66.866,-176.767,7.174,148.402
C09007=1200.361,283.814,-66.838,-176.771,7.172,148.402
C09008=1200.365,283.567,-66.809,-176.773,7.170,148.403
C09009=1200.370,283.318,-66.780,-176.775,7.167,148.403
C09010=1200.375,283.070,-66.751,-176.778,7.164,148.403
C09011=1200.378,282.822,-66.723,-176.780,7.161,148.403
C09012=1200.383,282.573,-66.694,-176.782,7.159,148.403
C09013=1200.388,282.325,-66.665,-176.786,7.157,148.403
C09014=1200.391,282.077,-66.637,-176.788,7.154,148.403
C09015=1200.396,281.828,-66.608,-176.790,7.151,148.403
C09016=1200.401,281.580,-66.579,-176.793,7.149,148.403
C09017=1200.404,281.332,-66.551,-176.795,7.146,148.403
C09018=1200.409,281.083,-66.523,-176.798,7.144,148.403
C09019=1200.413,280.835,-66.495,-176.801,7.141,148.404
C09020=1200.417,280.587,-66.465,-176.803,7.138,148.404
C09021=1200.422,280.338,-66.437,-176.805,7.136,148.404
C09022=1200.426,280.090,-66.409,-176.809,7.133,148.404
C09023=1200.431,279.841,-66.380,-176.811,7.131,148.404
C09024=1200.435,279.594,-66.352,-176.813,7.128,148.404
C09025=1200.439,279.345,-66.323,-176.816,7.126,148.404
C09026=1200.444,279.097,-66.295,-176.818,7.123,148.404
C09027=1200.448,278.848,-66.266,-176.821,7.121,148.404
C09028=1200.453,278.599,-66.238,-176.824,7.118,148.404
C09029=1200.457,278.352,-66.209,-176.826,7.116,148.404
C09030=1200.461,278.103,-66.180,-176.828,7.113,148.405
C09031=1200.465,277.855,-66.153,-176.831,7.111,148.405
C09032=1200.470,277.606,-66.124,-176.834,7.108,148.405
C09033=1200.474,277.358,-66.096,-176.836,7.106,148.405
C09034=1200.479,277.109,-66.067,-176.839,7.103,148.405
C09035=1200.483,276.862,-66.040,-176.841,7.101,148.405
C09036=1200.487,276.613,-66.011,-176.844,7.098,148.405
C09037=1200.491,276.364,-65.983,-176.846,7.096,148.405
C09038=1200.496,276.116,-65.955,-176.849,7.093,148.405
C09039=1200.500,275.867,-65.926,-176.851,7.091,148.406
C09040=1200.505,275.619,-65.898,-176.854,7.088,148.406
C09041=1200.509,275.371,-65.870,-176.856,7.086,148.406
C09042=1200.513,275.123,-65.842,-176.859,7.083,148.406
C09043=1200.518,274.874,-65.813,-176.862,7.081,148.406
C09044=1200.522,274.626,-65.785,-176.864,7.078,148.406
C09045=1200.526,274.377,-65.757,-176.866,7.076,148.406
C09046=1200.531,274.129,-65.729,-176.870,7.073,148.407
C09047=1200.535,273.881,-65.701,-176.872,7.071,148.407
C09048=1200.540,273.632,-65.672,-176.874,7.068,148.407
C09049=1200.544,273.384,-65.644,-176.877,7.066,148.407
C09050=1200.548,273.136,-65.616,-176.880,7.063,148.407
C09051=1200.553,272.888,-65.588,-176.882,7.061,148.407
C09052=1200.557,272.639,-65.560,-176.885,7.058,148.407
C09053=1200.561,272.391,-65.532,-176.887,7.056,148.407
C09054=1200.566,272.142,-65.504,-176.890,7.053,148.407
C09055=1200.570,271.894,-65.476,-176.892,7.051,148.407
C09056=1200.574,271.645,-65.448,-176.894,7.048,148.408
C09057=1200.579,271.397,-65.420,-176.897,7.046,148.408
C09058=1200.583,271.149,-65.392,-176.899,7.044,148.408
C09059=1200.588,270.900,-65.365,-176.902,7.041,148.408
C09060=1200.592,270.652,-65.337,-176.905,7.039,148.408
C09061=1200.596,270.403,-65.308,-176.908,7.036,148.408
C09062=1200.601,270.155,-65.280,-176.910,7.034,148.408
C09063=1200.604,269.907,-65.252,-176.913,7.031,148.409
C09064=1200.609,269.658,-65.225,-176.915,7.029,148.409
C09065=1200.614,269.410,-65.197,-176.918,7.026,148.409
C09066=1200.618,269.162,-65.169,-176.920,7.024,148.409
C09067=1200.623,268.913,-65.141,-176.923,7.021,148.409
C09068=1200.626,268.665,-65.113,-176.925,7.019,148.409
C09069=1200.631,268.416,-65.085,-176.928,7.017,148.409
C09070=1200.636,268.168,-65.058,-176.930,7.014,148.409
C09071=1200.640,267.919,-65.030,-176.933,7.012,148.410
C09072=1200.644,267.671,-65.002,-176.936,7.009,148.410
C09073=1200.649,267.423,-64.975,-176.938,7.007,148.410
C09074=1200.653,267.174,-64.946,-176.941,7.004,148.410
C09075=1200.658,266.926,-64.919,-176.943,7.002,148.410
C09076=1200.662,266.678,-64.891,-176.945,7.000,148.410
C09077=1200.666,266.429,-64.863,-176.948,6.997,148.410
C09078=1200.671,266.181,-64.836,-176.951,6.995,148.411
C09079=1200.675,265.933,-64.808,-176.953,6.992,148.411
C09080=1200.679,265.684,-64.781,-176.956,6.990,148.411
C09081=1200.684,265.435,-64.753,-176.959,6.987,148.411
C09082=1200.689,265.187,-64.725,-176.961,6.985,148.411
C09083=1200.693,264.938,-64.697,-176.964,6.983,148.411
C09084=1200.697,264.690,-64.670,-176.966,6.980,148.411
C09085=1200.702,264.442,-64.643,-176.968,6.978,148.412
C09086=1200.706,264.193,-64.615,-176.972,6.975,148.412
C09087=1200.710,263.945,-64.587,-176.974,6.973,148.412
C09088=1200.715,263.696,-64.560,-176.976,6.970,148.412
C09089=1200.719,263.448,-64.533,-176.979,6.968,148.412
C09090=1200.724,263.175,-64.503,-176.982,6.965,148.412
C09091=1200.729,262.902,-64.472,-176.984,6.963,148.413
C09092=1200.734,262.630,-64.442,-176.987,6.960,148.413
C09093=1200.739,262.356,-64.412,-176.990,6.957,148.413
C09094=1200.743,262.108,-64.385,-176.992,6.955,148.413
C09095=1200.748,261.860,-64.357,-176.996,6.953,148.413
C09096=1200.752,261.611,-64.330,-176.998,6.950,148.413
C09097=1200.756,261.362,-64.302,-177.001,6.948,148.414
C09098=1200.761,261.114,-64.275,-177.003,6.946,148.414
C09099=1200.765,260.866,-64.248,-177.005,6.943,148.414
C09100=1200.770,260.617,-64.221,-177.008,6.941,148.414
C09101=1200.774,260.369,-64.192,-177.011,6.939,148.414
C09102=1200.778,260.120,-64.165,-177.014,6.936,148.414
C09103=1200.783,259.872,-64.138,-177.016,6.934,148.414
C09104=1200.787,259.624,-64.112,-177.018,6.932,148.415
C09105=1200.791,259.376,-64.084,-177.021,6.929,148.415
C09106=1200.795,259.127,-64.057,-177.023,6.927,148.415
C09107=1200.800,258.878,-64.030,-177.026,6.925,148.415
C09108=1200.805,258.630,-64.003,-177.029,6.922,148.415
C09109=1200.809,258.381,-63.975,-177.031,6.920,148.416
C09110=1200.814,258.133,-63.948,-177.034,6.917,148.416
C09111=1200.818,257.884,-63.920,-177.036,6.915,148.416
C09112=1200.822,257.635,-63.893,-177.039,6.913,148.416
C09113=1200.827,257.387,-63.866,-177.042,6.910,148.416
C09114=1200.831,257.139,-63.840,-177.044,6.908,148.416
C09115=1200.836,256.890,-63.813,-177.046,6.906,148.416
C09116=1200.840,256.642,-63.786,-177.049,6.903,148.417
C09117=1200.845,256.393,-63.758,-177.052,6.901,148.417
C09118=1200.849,256.145,-63.730,-177.054,6.899,148.417
C09119=1200.853,255.896,-63.703,-177.057,6.896,148.417
C09120=1200.857,255.648,-63.677,-177.059,6.894,148.417
C09121=1200.862,255.400,-63.650,-177.062,6.891,148.418
C09122=1200.867,255.151,-63.623,-177.064,6.889,148.418
C09123=1200.871,254.903,-63.596,-177.067,6.887,148.418
C09124=1200.876,254.654,-63.569,-177.070,6.884,148.418
C09125=1200.880,254.406,-63.542,-177.072,6.882,148.418
C09126=1200.884,254.157,-63.515,-177.075,6.880,148.418
C09127=1200.888,253.908,-63.488,-177.078,6.878,148.419
C09128=1200.893,253.660,-63.461,-177.080,6.875,148.419
C09129=1200.897,253.412,-63.434,-177.083,6.874,148.419
C09130=1200.902,253.163,-63.407,-177.085,6.871,148.419
C09131=1200.907,252.914,-63.381,-177.088,6.869,148.419
C09132=1200.911,252.666,-63.354,-177.090,6.867,148.420
C09133=1200.915,252.417,-63.327,-177.093,6.864,148.420
C09134=1200.920,252.169,-63.300,-177.095,6.862,148.420
C09135=1200.925,251.920,-63.273,-177.098,6.860,148.420
C09136=1200.928,251.672,-63.247,-177.101,6.857,148.420
